RoboDK station: RobotCell.rdk

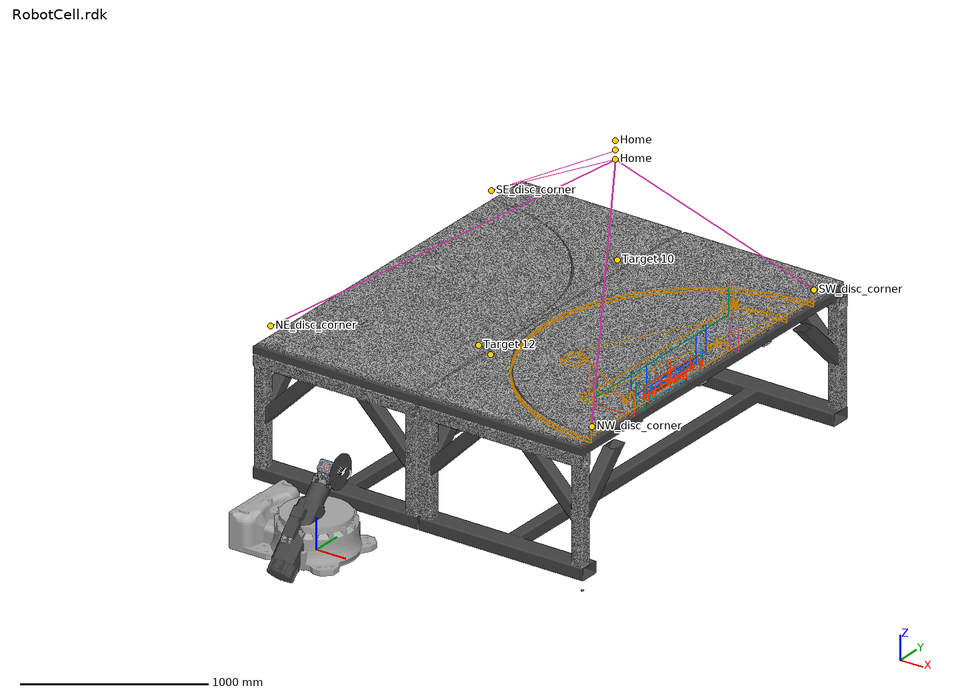
[picture v0: the station drawn from its stored meshes, robots at their saved joint values, targets as dots, program paths as lines]
Station RobotCell (saved by RoboDK 5.6.8). Poses are relative to the parent item; angles as X-Y-Z fixed-axis rotations.
  - frame Kawasaki BX130X Base at (0, 0, 0) mm
    - robot Kawasaki BX130X: 6 axes, payload 130 kg, reach 2991 mm, repeatability 0.06 mm, weight 920 kg
        joint limits [-160, -60, -75, -210, -125, -210] to [160, 76, 90, 210, 125, 210]; home [0, 0, 0, 0, 0, 0]; saved at [15.367, 30.588, 15.611, 20.856, -32.878, -29.669]
      - tool Bare Spindle, TCP at (-2.41, 51.17, 373.7) mm, rotated rx 0.82 ry 46.22 rz 88.69 deg
      - tool Sawblade, TCP at (72.1, 194.8, 514.4) mm, rotated rx 1 ry 44.99 rz 91.98 deg, size 476.9 x 3677.1 x 608 mm, geometry from Sawblade.step
      - tool halfInchUpcut, TCP at (-1.57, 133.94, 455.3) mm, rotated rx 0 ry 45 rz 90 deg, size 451 x 3595 x 525.8 mm, geometry from halfInchUpcut.step
  - frame Work hold down at (0, 0, -2) mm
  - folder FrontWallWest
    - machining project Blade_door_east: C:/Users/kris/AppData/Local/Temp/Front wall cutout v15.apt:2 | rotZ(0) | rotX(0)*rotY(0) | rotz(0) | onStart | onPathStart | onApproach | onPoint | onRetract | onFinish | Extruder(%1) | default | default | OutOnMov(%1) | OutOffMov(%1) | onPathFinish | M_RunCode(%1)
    - machining project Blade_doorframe_east: C:/Users/kris/AppData/Local/Temp/Front wall cutout v15.apt | rotZ(0) | rotX(0)*rotY(0) | rotz(0) | onStart | onPathStart | onApproach | onPoint | onRetract | onFinish | Extruder(%1) | default | default | OutOnMov(%1) | OutOffMov(%1) | onPathFinish | M_RunCode(%1)
    - machining project Blade_doorwindow_east: C:/Users/kris/AppData/Local/Temp/Front wall cutout v11.apt:3 | rotZ(0) | rotX(0)*rotY(0) | rotz(0) | onStart | onPathStart | onApproach | onPoint | onRetract | onFinish | Extruder(%1) | default | default | OutOnMov(%1) | OutOffMov(%1) | onPathFinish | M_RunCode(%1)
    - machining project Blade_door_north: C:/Users/kris/AppData/Local/Temp/Front wall cutout v11.apt:4 | rotZ(0) | rotX(0)*rotY(0) | rotz(0) | onStart | onPathStart | onApproach | onPoint | onRetract | onFinish | Extruder(%1) | default | default | OutOnMov(%1) | OutOffMov(%1) | onPathFinish | M_RunCode(%1)
    - machining project Blade_window_north: C:/Users/kris/AppData/Local/Temp/Front wall cutout v11.apt:5 | rotZ(0) | rotX(0)*rotY(0) | rotz(0) | onStart | onPathStart | onApproach | onPoint | onRetract | onFinish | Extruder(%1) | default | default | OutOnMov(%1) | OutOffMov(%1) | onPathFinish | M_RunCode(%1)
    - machining project Blade_window_south: C:/Users/kris/AppData/Local/Temp/Front wall cutout v11.apt:6 | rotZ(0) | rotX(0)*rotY(0) | rotz(0) | onStart | onPathStart | onApproach | onPoint | onRetract | onFinish | Extruder(%1) | default | default | OutOnMov(%1) | OutOffMov(%1) | onPathFinish | M_RunCode(%1)
    - machining project Roughing: C:/Users/kris/AppData/Local/Temp/Front wall cutout v11.apt:7 | rotZ(0) | rotX(0)*rotY(0) | rotZ(0)
    - machining project Blade_handles_west: C:/Users/kris/AppData/Local/Temp/Front wall cutout v12.apt | rotZ(0) | rotX(0)*rotY(0) | rotz(0) | onStart | onPathStart | onApproach | onPoint | onRetract | onFinish | Extruder(%1) | default | default | OutOnMov(%1) | OutOffMov(%1) | onPathFinish | M_RunCode(%1)
    - machining project Blade_handles_east: C:/Users/kris/AppData/Local/Temp/Front wall cutout v12.apt:2 | rotZ(0) | rotX(0)*rotY(0) | rotz(0) | onStart | onPathStart | onApproach | onPoint | onRetract | onFinish | Extruder(%1) | default | default | OutOnMov(%1) | OutOffMov(%1) | onPathFinish | M_RunCode(%1)
    - machining project Handles_roughing: C:/Users/kris/AppData/Local/Temp/Front wall cutout v12.apt:3 | rotZ(0) | rotX(0)*rotY(0) | rotZ(0) | onStart | onPathStart | onApproach | onPoint | onRetract | onFinish | Extruder(%1) | default | default | OutOnMov(%1) | OutOffMov(%1) | onPathFinish | M_RunCode(%1)
    - program Blade_doorwindow_east (21 instructions, listed below)
    - program Blade_door_north (21 instructions, listed below)
    - program Blade_window_north (21 instructions, listed below)
    - program Blade_window_south (21 instructions, listed below)
    - program Roughing (2440 instructions, listed below)
    - program Blade_handles_west (25 instructions, listed below)
    - program Blade_handles_east (22 instructions, listed below)
    - program Handles_roughing (174 instructions, listed below)
    - program Blade_door_east (20 instructions, listed below)
  - object Front wall cutout v15 at (0, 0, 0) mm, size 2167.6 x 2462.4 x 856 mm, geometry from Front wall cutout v15.step
  - frame CalibrationFrame at (0, 0, 0) mm
    - target Home (Cartesian target) at (0.67, 2769.12, 1198.75) mm, rotated rx -177.74 ry 28.55 rz -88.97 deg; joints [-0.25, 14.674, 2.172, -12.213, -4.012, 10.365] of Kawasaki BX130X
    - target SW_disc_corner (Cartesian target) at (1075.28, 3073.73, 606.29) mm, rotated rx 180 ry 0 rz -88.75 deg; joints [21.99, 63.467, 60.14, 22.667, -46.398, -32.962] of Kawasaki BX130X
    - target Home (Cartesian target) at (0.67, 2769.12, 1198.75) mm, rotated rx -177.74 ry 28.55 rz -88.97 deg; joints [-0.25, 14.674, 2.172, -12.213, -4.012, 10.365] of Kawasaki BX130X
    - target NW_disc_corner (Cartesian target) at (1057.37, 1041.81, 606.29) mm, rotated rx 180 ry 0 rz -88.75 deg; joints [58.442, -29.711, -49.966, 48.514, -54.582, -83.664] of Kawasaki BX130X
    - target Home (Cartesian target) at (0.67, 2769.12, 1198.75) mm, rotated rx -177.74 ry 28.55 rz -88.97 deg; joints [-0.25, 14.674, 2.172, -12.213, -4.012, 10.365] of Kawasaki BX130X
    - target NE_disc_corner (Cartesian target) at (-1038.05, 1060.27, 606.29) mm, rotated rx -180 ry 0 rz -88.75 deg; joints [-56.747, -31.242, -50.944, 132.324, 52.01, -100.14] of Kawasaki BX130X
    - target Home (Cartesian target) at (0.67, 2769.12, 1198.75) mm, rotated rx -177.74 ry 28.55 rz -88.97 deg; joints [-0.25, 14.674, 2.172, -12.213, -4.012, 10.365] of Kawasaki BX130X
    - target SE_disc_corner (Cartesian target) at (-1020.25, 3079.49, 606.29) mm, rotated rx 180 ry 0 rz -88.75 deg; joints [-20.561, 60.823, 55.864, 160.128, 43.451, -151.385] of Kawasaki BX130X
    - target Home (Cartesian target) at (0.67, 2769.12, 1253.75) mm, rotated rx -177.74 ry 28.55 rz -88.97 deg; joints [-0.25, 14.499, 3.862, -8.354, -5.848, 6.491] of Kawasaki BX130X
    - target Target 10 (Cartesian target) at (10.17, 2770.62, 606.29) mm, rotated rx -180 ry 0 rz -90 deg; joints [0.282, 28.794, 8.219, 0.482, -24.427, -0.639] of Kawasaki BX130X
    - target Home (Cartesian target) at (0.67, 2769.12, 1253.75) mm, rotated rx -177.74 ry 28.55 rz -88.97 deg; joints [-0.25, 14.499, 3.862, -8.354, -5.848, 6.491] of Kawasaki BX130X
    - target Target 12 (Cartesian target) at (-1.2, 1504.96, 606.29) mm, rotated rx 180 ry 0 rz -88.97 deg; joints [0.375, -38.885, -55.483, 2.09, -28.427, -2.833] of Kawasaki BX130X
    - target Home (Cartesian target) at (0.67, 2769.12, 1308.75) mm, rotated rx -177.74 ry 28.55 rz -88.97 deg; joints [-0.25, 14.413, 5.654, -6.334, -7.711, 4.458] of Kawasaki BX130X
    - target Target 14 (Cartesian target) at (114.89, 1450.3, 606.29) mm, rotated rx 180 ry 0 rz -88.97 deg; joints [6.616, -42.397, -57.387, 10.621, -30.699, -14.583] of Kawasaki BX130X
  - program checkTableCalibration (11 instructions, listed below)
  - program Blade_doorframe_east (24 instructions, listed below)
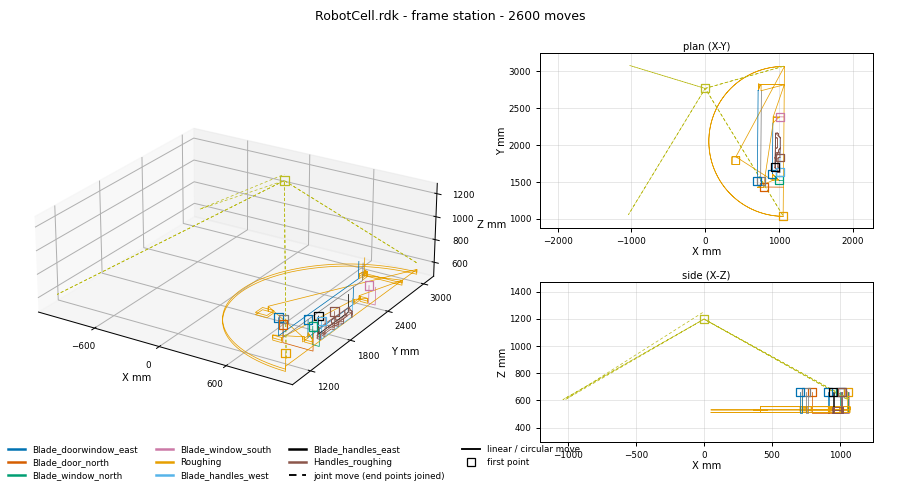
[picture p0: tool path of RobotCell.rdk in frame station, 2600 of 2600 moves have a stored position in this frame; points joined in program order, loops and branches not executed]

--- program Blade_doorwindow_east (robot Kawasaki BX130X) ---
  Smooth(1)
  Set speed (100.0 mm/s)
  Set Ref.: Work hold down
  Set Tool: Sawblade
  Show Sawblade
  MoveJ 1 to (911.47, 1609.21, 666.29) mm, rotated rx 180 ry 0 rz -90.5 deg; joints [34.508, -17.696, -36.382, 39.95, -39.175, -59.907]
  MoveL 2 to (911.47, 1609.21, 666.29) mm, rotated rx 180 ry 0 rz -90.5 deg; joints [34.508, -17.696, -36.382, 39.95, -39.175, -59.907]
  MoveL 3 to (911.47, 1609.21, 566.29) mm, rotated rx 180 ry 0 rz -90.5 deg; joints [34.508, -16.451, -38.924, 43.196, -36.34, -64.01]
  MoveL 4 to (911.47, 1609.21, 566.29) mm, rotated rx 180 ry 0 rz -90.5 deg; joints [34.508, -16.451, -38.924, 43.196, -36.34, -64.01]
  Set speed (100.0 mm/s)
  MoveL 5 to (911.47, 1609.21, 556.29) mm, rotated rx -180 ry 0 rz -90.5 deg; joints [34.508, -16.304, -39.162, 43.558, -36.06, -64.458]
  Set speed (5.6 mm/s)
  MoveL 6 to (911.47, 1609.21, 551.89) mm, rotated rx -180 ry 0 rz -90.5 deg; joints [34.508, -16.239, -39.266, 43.719, -35.937, -64.658]
  MoveL 7 to (911.47, 1609.21, 513.19) mm, rotated rx 180 ry 0 rz -90.5 deg; joints [34.508, -15.625, -40.158, 45.203, -34.863, -66.478]
  Set speed (133.3 mm/s)
  MoveL 8 to (917.55, 2299.44, 513.19) mm, rotated rx -180 ry 0 rz -90.5 deg; joints [23.876, 14.834, -9.851, 37.999, -28.292, -52.853]
  Set speed (100.0 mm/s)
  MoveL 9 to (917.55, 2299.44, 566.29) mm, rotated rx -180 ry 0 rz -90.5 deg; joints [23.876, 14.117, -8.799, 36.076, -29.704, -50.655]
  MoveL 10 to (917.55, 2299.44, 566.29) mm, rotated rx -180 ry 0 rz -90.5 deg; joints [23.876, 14.117, -8.799, 36.076, -29.704, -50.655]
  MoveL 11 to (917.55, 2299.44, 666.29) mm, rotated rx 180 ry 0 rz -90.5 deg; joints [23.876, 12.98, -6.592, 32.933, -32.461, -46.986]
  Print: /'Blade door top'

--- program Blade_door_north (robot Kawasaki BX130X) ---
  Smooth(1)
  Set speed (100.0 mm/s)
  Set Ref.: Work hold down
  Set Tool: Sawblade
  Show Sawblade
  MoveJ 1 to (794.89, 1433.16, 666.29) mm, rotated rx -180 ry 0 rz 179.5 deg; joints [15.202, -13.662, -33.122, -48.467, -65.42, 92.913]
  MoveL 2 to (794.89, 1433.16, 666.29) mm, rotated rx -180 ry 0 rz 179.5 deg; joints [15.202, -13.662, -33.122, -48.467, -65.42, 92.913]
  MoveL 3 to (794.89, 1433.16, 566.29) mm, rotated rx 180 ry 0 rz 179.5 deg; joints [15.202, -12.385, -35.587, -49.836, -62.972, 96.057]
  MoveL 4 to (794.89, 1433.16, 566.29) mm, rotated rx 180 ry 0 rz 179.5 deg; joints [15.202, -12.385, -35.587, -49.836, -62.972, 96.057]
  Set speed (100.0 mm/s)
  MoveL 5 to (794.89, 1433.16, 556.29) mm, rotated rx -180 ry 0 rz 179.5 deg; joints [15.202, -12.236, -35.818, -49.985, -62.728, 96.384]
  Set speed (5.6 mm/s)
  MoveL 6 to (794.89, 1433.16, 551.89) mm, rotated rx -180 ry 0 rz 179.5 deg; joints [15.202, -12.169, -35.918, -50.052, -62.62, 96.528]
  MoveL 7 to (794.89, 1433.16, 513.19) mm, rotated rx -180 ry 0 rz 179.5 deg; joints [15.202, -11.55, -36.78, -50.654, -61.675, 97.818]
  Set speed (133.3 mm/s)
  MoveL 8 to (1060.8, 1430.82, 513.19) mm, rotated rx -180 ry 0 rz 179.5 deg; joints [24.193, -6.922, -32.695, -51.648, -55.011, 92.337]
  Set speed (100.0 mm/s)
  MoveL 9 to (1060.8, 1430.82, 566.29) mm, rotated rx -180 ry 0 rz 179.5 deg; joints [24.193, -7.755, -31.542, -50.591, -56.258, 90.464]
  MoveL 10 to (1060.8, 1430.82, 566.29) mm, rotated rx -180 ry 0 rz 179.5 deg; joints [24.193, -7.755, -31.542, -50.591, -56.258, 90.464]
  MoveL 11 to (1060.8, 1430.82, 666.29) mm, rotated rx -180 ry 0 rz 179.5 deg; joints [24.193, -9.049, -29.155, -48.799, -58.64, 87.134]
  Print: /'Blade door window top'

--- program Blade_window_north (robot Kawasaki BX130X) ---
  Smooth(1)
  Set speed (100.0 mm/s)
  Set Ref.: Work hold down
  Set Tool: Sawblade
  Show Sawblade
  MoveJ 1 to (1002.24, 1523.24, 666.29) mm, rotated rx -180 ry 0 rz 179.5 deg; joints [21.13, -5.832, -26.235, -48.977, -60.608, 89.581]
  MoveL 2 to (1002.24, 1523.24, 666.29) mm, rotated rx -180 ry 0 rz 179.5 deg; joints [21.13, -5.832, -26.235, -48.977, -60.608, 89.581]
  MoveL 3 to (1002.24, 1523.24, 566.29) mm, rotated rx -180 ry 0 rz 179.5 deg; joints [21.13, -4.54, -28.576, -50.616, -58.262, 92.804]
  MoveL 4 to (1002.24, 1523.24, 566.29) mm, rotated rx -180 ry 0 rz 179.5 deg; joints [21.13, -4.54, -28.576, -50.616, -58.262, 92.804]
  Set speed (100.0 mm/s)
  MoveL 5 to (1002.24, 1523.24, 556.29) mm, rotated rx -180 ry 0 rz 179.5 deg; joints [21.13, -4.392, -28.794, -50.793, -58.03, 93.138]
  Set speed (5.6 mm/s)
  MoveL 6 to (1002.24, 1523.24, 551.89) mm, rotated rx 180 ry 0 rz 179.5 deg; joints [21.13, -4.325, -28.89, -50.871, -57.928, 93.286]
  MoveL 7 to (1002.24, 1523.24, 513.19) mm, rotated rx -180 ry 0 rz 179.5 deg; joints [21.13, -3.713, -29.703, -51.58, -57.035, 94.604]
  Set speed (133.3 mm/s)
  MoveL 8 to (1061.61, 1522.72, 513.19) mm, rotated rx 180 ry 0 rz 179.5 deg; joints [22.97, -2.615, -28.649, -51.728, -55.71, 93.414]
  Set speed (100.0 mm/s)
  MoveL 9 to (1061.61, 1522.72, 566.29) mm, rotated rx 180 ry 0 rz 179.5 deg; joints [22.97, -3.438, -27.529, -50.718, -56.927, 91.594]
  MoveL 10 to (1061.61, 1522.72, 566.29) mm, rotated rx 180 ry 0 rz 179.5 deg; joints [22.97, -3.438, -27.529, -50.718, -56.927, 91.594]
  MoveL 11 to (1061.61, 1522.72, 666.29) mm, rotated rx 180 ry 0 rz 179.5 deg; joints [22.97, -4.728, -25.203, -48.996, -59.259, 88.337]
  Print: /'Blade door window south'

--- program Blade_window_south (robot Kawasaki BX130X) ---
  Smooth(1)
  Set speed (100.0 mm/s)
  Set Ref.: Work hold down
  Set Tool: Sawblade
  Show Sawblade
  MoveJ 1 to (1009.82, 2383.81, 666.29) mm, rotated rx -180 ry 0 rz 179.49 deg; joints [14.255, 35.484, 22.375, -46.548, -70.389, 88.528]
  MoveL 2 to (1009.82, 2383.81, 666.29) mm, rotated rx -180 ry 0 rz 179.49 deg; joints [14.255, 35.484, 22.375, -46.548, -70.389, 88.528]
  MoveL 3 to (1009.82, 2383.81, 566.29) mm, rotated rx -180 ry 0 rz 179.49 deg; joints [14.255, 36.15, 19.85, -47.43, -68.212, 91.022]
  MoveL 4 to (1009.82, 2383.81, 566.29) mm, rotated rx -180 ry 0 rz 179.49 deg; joints [14.255, 36.15, 19.85, -47.43, -68.212, 91.022]
  Set speed (100.0 mm/s)
  MoveL 5 to (1009.82, 2383.81, 556.29) mm, rotated rx -180 ry 0 rz 179.49 deg; joints [14.255, 36.232, 19.62, -47.522, -68, 91.271]
  Set speed (5.6 mm/s)
  MoveL 6 to (1009.82, 2383.81, 551.89) mm, rotated rx -180 ry 0 rz 179.49 deg; joints [14.255, 36.27, 19.519, -47.563, -67.907, 91.381]
  MoveL 7 to (1009.82, 2383.81, 513.19) mm, rotated rx -180 ry 0 rz 179.49 deg; joints [14.255, 36.621, 18.668, -47.932, -67.099, 92.344]
  Set speed (133.3 mm/s)
  MoveL 8 to (1069.19, 2383.28, 513.19) mm, rotated rx -180 ry 0 rz 179.49 deg; joints [15.552, 37.428, 19.819, -47.863, -66.413, 91.165]
  Set speed (100.0 mm/s)
  MoveL 9 to (1069.19, 2383.28, 566.29) mm, rotated rx 180 ry 0 rz 179.49 deg; joints [15.552, 36.97, 21.014, -47.344, -67.527, 89.838]
  MoveL 10 to (1069.19, 2383.28, 566.29) mm, rotated rx 180 ry 0 rz 179.49 deg; joints [15.552, 36.97, 21.014, -47.344, -67.527, 89.838]
  MoveL 11 to (1069.19, 2383.28, 666.29) mm, rotated rx -180 ry 0 rz 179.49 deg; joints [15.552, 36.33, 23.568, -46.431, -69.711, 87.335]
  Print: /'Roughing'

--- program Roughing (robot Kawasaki BX130X) ---
  Smooth(1)
  Set speed (100.0 mm/s)
  Set Ref.: Work hold down
  Set Tool: halfInchUpcut
  Show halfInchUpcut
  MoveJ 1 to (1057.31, 1035.46, 666.29) mm, rotated rx -180 ry 0 rz -88.32 deg; joints [58.753, -30.506, -48.445, 47.413, -56.648, -82.141]
  MoveL 2 to (1057.31, 1035.46, 666.29) mm, rotated rx -180 ry 0 rz -88.32 deg; joints [58.753, -30.506, -48.445, 47.413, -56.648, -82.141]
  MoveL 3 to (1057.31, 1035.46, 566.29) mm, rotated rx 180 ry 0 rz -88.32 deg; joints [58.753, -29.128, -51.071, 49.488, -53.99, -85.786]
  MoveL 4 to (1057.31, 1035.46, 566.29) mm, rotated rx 180 ry 0 rz -88.32 deg; joints [58.753, -29.128, -51.071, 49.488, -53.99, -85.786]
  Set speed (100.0 mm/s)
  MoveL 5 to (1057.31, 1035.46, 556.29) mm, rotated rx -180 ry 0 rz -88.32 deg; joints [58.753, -28.961, -51.317, 49.718, -53.723, -86.175]
  Set speed (5.6 mm/s)
  MoveL 6 to (1057.31, 1035.46, 552.29) mm, rotated rx -180 ry 0 rz -88.32 deg; joints [58.753, -28.893, -51.415, 49.811, -53.616, -86.332]
  MoveL 7 to (1057.31, 1035.46, 532.29) mm, rotated rx 180 ry 0 rz -88.32 deg; joints [58.753, -28.539, -51.896, 50.287, -53.08, -87.13]
  Set speed (91.9 mm/s)
  MoveL 8 to (1054.46, 1035.49, 532.29) mm, rotated rx 180 ry 0 rz -88.32 deg; joints [58.684, -28.699, -52.001, 50.252, -53.066, -87.026]
  MoveL 9 to (1051.61, 1035.53, 532.29) mm, rotated rx -180 ry 0 rz -88.32 deg; joints [58.614, -28.86, -52.105, 50.217, -53.053, -86.921]
  MoveL 10 to (1048.77, 1035.57, 532.29) mm, rotated rx 180 ry 0 rz -88.32 deg; joints [58.544, -29.02, -52.209, 50.181, -53.039, -86.816]
  MoveL 11 to (1045.92, 1035.62, 532.29) mm, rotated rx -180 ry 0 rz -88.32 deg; joints [58.473, -29.18, -52.313, 50.145, -53.025, -86.71]
  MoveL 12 to (1043.07, 1035.69, 532.29) mm, rotated rx -180 ry 0 rz -88.32 deg; joints [58.402, -29.34, -52.417, 50.109, -53.011, -86.603]
  MoveL 13 to (1040.22, 1035.75, 532.29) mm, rotated rx -180 ry 0 rz -88.32 deg; joints [58.33, -29.5, -52.52, 50.072, -52.997, -86.495]
  MoveL 14 to (1037.37, 1035.83, 532.29) mm, rotated rx -180 ry 0 rz -88.32 deg; joints [58.258, -29.659, -52.623, 50.035, -52.982, -86.387]
  MoveL 15 to (1034.52, 1035.92, 532.29) mm, rotated rx -180 ry 0 rz -88.32 deg; joints [58.185, -29.819, -52.726, 49.998, -52.967, -86.278]
  MoveL 16 to (1031.67, 1036.01, 532.29) mm, rotated rx 180 ry 0 rz -88.32 deg; joints [58.111, -29.978, -52.828, 49.961, -52.952, -86.169]
  MoveL 17 to (1028.82, 1036.11, 532.29) mm, rotated rx 180 ry 0 rz -88.32 deg; joints [58.037, -30.138, -52.93, 49.923, -52.937, -86.058]
  MoveL 18 to (1025.98, 1036.22, 532.29) mm, rotated rx 180 ry 0 rz -88.32 deg; joints [57.962, -30.297, -53.031, 49.885, -52.921, -85.947]
  MoveL 19 to (1023.13, 1036.34, 532.29) mm, rotated rx 180 ry 0 rz -88.32 deg; joints [57.887, -30.456, -53.132, 49.847, -52.906, -85.836]
  MoveL 20 to (1020.28, 1036.46, 532.29) mm, rotated rx -180 ry 0 rz -88.32 deg; joints [57.811, -30.615, -53.233, 49.808, -52.889, -85.723]
  MoveL 21 to (1017.43, 1036.6, 532.29) mm, rotated rx 180 ry 0 rz -88.32 deg; joints [57.734, -30.774, -53.334, 49.769, -52.873, -85.61]
  MoveL 22 to (1014.59, 1036.74, 532.29) mm, rotated rx -180 ry 0 rz -88.32 deg; joints [57.657, -30.933, -53.434, 49.73, -52.857, -85.496]
  MoveL 23 to (1011.74, 1036.89, 532.29) mm, rotated rx -180 ry 0 rz -88.32 deg; joints [57.579, -31.092, -53.534, 49.691, -52.84, -85.381]
  MoveL 24 to (1008.9, 1037.04, 532.29) mm, rotated rx -180 ry 0 rz -88.32 deg; joints [57.501, -31.25, -53.633, 49.651, -52.823, -85.266]
  MoveL 25 to (1006.05, 1037.21, 532.29) mm, rotated rx -180 ry 0 rz -88.32 deg; joints [57.422, -31.409, -53.733, 49.611, -52.805, -85.15]
  MoveL 26 to (1003.21, 1037.38, 532.29) mm, rotated rx 180 ry 0 rz -88.32 deg; joints [57.342, -31.567, -53.831, 49.57, -52.788, -85.033]
  MoveL 27 to (1000.36, 1037.56, 532.29) mm, rotated rx -180 ry 0 rz -88.32 deg; joints [57.262, -31.725, -53.93, 49.53, -52.77, -84.916]
  MoveL 28 to (997.52, 1037.75, 532.29) mm, rotated rx -180 ry 0 rz -88.32 deg; joints [57.181, -31.883, -54.028, 49.489, -52.752, -84.798]
  MoveL 29 to (994.68, 1037.95, 532.29) mm, rotated rx -180 ry 0 rz -88.32 deg; joints [57.099, -32.04, -54.126, 49.447, -52.733, -84.679]
  MoveL 30 to (991.83, 1038.15, 532.29) mm, rotated rx -180 ry 0 rz -88.32 deg; joints [57.017, -32.198, -54.223, 49.406, -52.715, -84.559]
  MoveL 31 to (988.99, 1038.36, 532.29) mm, rotated rx 180 ry 0 rz -88.32 deg; joints [56.935, -32.355, -54.32, 49.364, -52.696, -84.439]
  MoveL 32 to (986.15, 1038.58, 532.29) mm, rotated rx 180 ry 0 rz -88.32 deg; joints [56.851, -32.512, -54.417, 49.322, -52.676, -84.318]
  MoveL 33 to (983.31, 1038.81, 532.29) mm, rotated rx 180 ry 0 rz -88.32 deg; joints [56.767, -32.669, -54.513, 49.279, -52.657, -84.196]
  MoveL 34 to (980.47, 1039.05, 532.29) mm, rotated rx -180 ry 0 rz -88.32 deg; joints [56.683, -32.826, -54.609, 49.236, -52.637, -84.074]
  MoveL 35 to (977.63, 1039.29, 532.29) mm, rotated rx 180 ry 0 rz -88.32 deg; joints [56.598, -32.982, -54.704, 49.193, -52.617, -83.951]
  MoveL 36 to (974.79, 1039.55, 532.29) mm, rotated rx 180 ry 0 rz -88.32 deg; joints [56.512, -33.139, -54.8, 49.15, -52.597, -83.827]
  MoveL 37 to (971.95, 1039.81, 532.29) mm, rotated rx 180 ry 0 rz -88.32 deg; joints [56.425, -33.295, -54.894, 49.106, -52.576, -83.702]
  MoveL 38 to (969.12, 1040.08, 532.29) mm, rotated rx -180 ry 0 rz -88.32 deg; joints [56.338, -33.451, -54.989, 49.062, -52.555, -83.577]
  MoveL 39 to (966.28, 1040.35, 532.29) mm, rotated rx -180 ry 0 rz -88.32 deg; joints [56.251, -33.606, -55.083, 49.017, -52.534, -83.451]
  MoveL 40 to (963.44, 1040.64, 532.29) mm, rotated rx 180 ry 0 rz -88.32 deg; joints [56.162, -33.762, -55.176, 48.973, -52.512, -83.325]
  MoveL 41 to (960.61, 1040.93, 532.29) mm, rotated rx -180 ry 0 rz -88.32 deg; joints [56.073, -33.917, -55.27, 48.928, -52.49, -83.197]
  MoveL 42 to (957.78, 1041.23, 532.29) mm, rotated rx -180 ry 0 rz -88.32 deg; joints [55.984, -34.072, -55.363, 48.882, -52.468, -83.069]
  MoveL 43 to (954.94, 1041.54, 532.29) mm, rotated rx 180 ry 0 rz -88.32 deg; joints [55.894, -34.226, -55.455, 48.836, -52.446, -82.94]
  MoveL 44 to (952.11, 1041.85, 532.29) mm, rotated rx 180 ry 0 rz -88.32 deg; joints [55.803, -34.381, -55.547, 48.79, -52.423, -82.811]
  MoveL 45 to (949.28, 1042.18, 532.29) mm, rotated rx 180 ry 0 rz -88.32 deg; joints [55.711, -34.535, -55.639, 48.744, -52.4, -82.681]
  MoveL 46 to (946.45, 1042.51, 532.29) mm, rotated rx 180 ry 0 rz -88.32 deg; joints [55.619, -34.688, -55.73, 48.697, -52.376, -82.55]
  MoveL 47 to (943.62, 1042.85, 532.29) mm, rotated rx -180 ry 0 rz -88.32 deg; joints [55.526, -34.842, -55.821, 48.65, -52.353, -82.418]
  MoveL 48 to (940.79, 1043.2, 532.29) mm, rotated rx -180 ry 0 rz -88.32 deg; joints [55.433, -34.995, -55.912, 48.603, -52.329, -82.286]
  MoveL 49 to (937.96, 1043.56, 532.29) mm, rotated rx -180 ry 0 rz -88.32 deg; joints [55.339, -35.148, -56.002, 48.555, -52.304, -82.153]
  MoveL 50 to (935.14, 1043.92, 532.29) mm, rotated rx 180 ry 0 rz -88.32 deg; joints [55.244, -35.301, -56.092, 48.507, -52.28, -82.02]
  MoveL 51 to (932.31, 1044.29, 532.29) mm, rotated rx -180 ry 0 rz -88.32 deg; joints [55.149, -35.453, -56.181, 48.458, -52.255, -81.885]
  MoveL 52 to (929.49, 1044.67, 532.29) mm, rotated rx -180 ry 0 rz -88.32 deg; joints [55.053, -35.605, -56.27, 48.41, -52.229, -81.75]
  MoveL 53 to (926.66, 1045.06, 532.29) mm, rotated rx -180 ry 0 rz -88.32 deg; joints [54.956, -35.757, -56.358, 48.361, -52.204, -81.615]
  MoveL 54 to (923.84, 1045.45, 532.29) mm, rotated rx -180 ry 0 rz -88.32 deg; joints [54.859, -35.908, -56.447, 48.311, -52.178, -81.478]
  MoveL 55 to (921.02, 1045.86, 532.29) mm, rotated rx 180 ry 0 rz -88.32 deg; joints [54.761, -36.059, -56.534, 48.261, -52.151, -81.341]
  MoveL 56 to (918.2, 1046.27, 532.29) mm, rotated rx 180 ry 0 rz -88.32 deg; joints [54.663, -36.21, -56.622, 48.211, -52.125, -81.203]
  MoveL 57 to (915.38, 1046.69, 532.29) mm, rotated rx 180 ry 0 rz -88.32 deg; joints [54.563, -36.36, -56.708, 48.161, -52.098, -81.065]
  MoveL 58 to (912.56, 1047.11, 532.29) mm, rotated rx 180 ry 0 rz -88.32 deg; joints [54.464, -36.51, -56.795, 48.11, -52.07, -80.926]
  MoveL 59 to (909.75, 1047.55, 532.29) mm, rotated rx 180 ry 0 rz -88.32 deg; joints [54.363, -36.659, -56.881, 48.059, -52.043, -80.786]
  MoveL 60 to (906.93, 1047.99, 532.29) mm, rotated rx 180 ry 0 rz -88.32 deg; joints [54.262, -36.809, -56.967, 48.007, -52.015, -80.646]
  MoveL 61 to (904.12, 1048.44, 532.29) mm, rotated rx -180 ry 0 rz -88.32 deg; joints [54.16, -36.957, -57.052, 47.955, -51.986, -80.504]
  MoveL 62 to (901.31, 1048.9, 532.29) mm, rotated rx 180 ry 0 rz -88.32 deg; joints [54.058, -37.106, -57.136, 47.903, -51.957, -80.363]
  MoveL 63 to (898.49, 1049.37, 532.29) mm, rotated rx -180 ry 0 rz -88.32 deg; joints [53.955, -37.254, -57.221, 47.851, -51.928, -80.22]
  MoveL 64 to (895.68, 1049.84, 532.29) mm, rotated rx -180 ry 0 rz -88.32 deg; joints [53.851, -37.401, -57.305, 47.798, -51.899, -80.077]
  MoveL 65 to (892.87, 1050.33, 532.29) mm, rotated rx 180 ry 0 rz -88.32 deg; joints [53.747, -37.549, -57.388, 47.744, -51.869, -79.933]
  MoveL 66 to (890.07, 1050.82, 532.29) mm, rotated rx -180 ry 0 rz -88.32 deg; joints [53.641, -37.695, -57.471, 47.691, -51.839, -79.789]
  MoveL 67 to (887.26, 1051.31, 532.29) mm, rotated rx 180 ry 0 rz -88.32 deg; joints [53.536, -37.842, -57.554, 47.637, -51.808, -79.643]
  MoveL 68 to (884.46, 1051.82, 532.29) mm, rotated rx 180 ry 0 rz -88.32 deg; joints [53.429, -37.988, -57.636, 47.582, -51.777, -79.497]
  MoveL 69 to (881.65, 1052.33, 532.29) mm, rotated rx 180 ry 0 rz -88.32 deg; joints [53.322, -38.133, -57.718, 47.527, -51.746, -79.351]
  MoveL 70 to (878.85, 1052.86, 532.29) mm, rotated rx -180 ry 0 rz -88.32 deg; joints [53.215, -38.278, -57.799, 47.472, -51.714, -79.204]
  MoveL 71 to (876.05, 1053.39, 532.29) mm, rotated rx 180 ry 0 rz -88.32 deg; joints [53.106, -38.422, -57.88, 47.417, -51.682, -79.056]
  MoveL 72 to (873.25, 1053.92, 532.29) mm, rotated rx 180 ry 0 rz -88.32 deg; joints [52.998, -38.567, -57.96, 47.361, -51.649, -78.908]
  MoveL 73 to (870.46, 1054.47, 532.29) mm, rotated rx -180 ry 0 rz -88.32 deg; joints [52.888, -38.71, -58.04, 47.305, -51.617, -78.758]
  MoveL 74 to (867.66, 1055.02, 532.29) mm, rotated rx -180 ry 0 rz -88.32 deg; joints [52.778, -38.853, -58.119, 47.248, -51.583, -78.609]
  MoveL 75 to (864.87, 1055.58, 532.29) mm, rotated rx -180 ry 0 rz -88.32 deg; joints [52.667, -38.996, -58.198, 47.191, -51.55, -78.458]
  MoveL 76 to (862.07, 1056.15, 532.29) mm, rotated rx 180 ry 0 rz -88.32 deg; joints [52.555, -39.138, -58.277, 47.134, -51.516, -78.307]
  MoveL 77 to (859.28, 1056.73, 532.29) mm, rotated rx -180 ry 0 rz -88.32 deg; joints [52.443, -39.279, -58.355, 47.076, -51.481, -78.156]
  MoveL 78 to (856.49, 1057.31, 532.29) mm, rotated rx 180 ry 0 rz -88.32 deg; joints [52.33, -39.42, -58.432, 47.018, -51.446, -78.003]
  MoveL 79 to (853.71, 1057.91, 532.29) mm, rotated rx 180 ry 0 rz -88.32 deg; joints [52.217, -39.561, -58.509, 46.96, -51.411, -77.85]
  MoveL 80 to (850.92, 1058.51, 532.29) mm, rotated rx 180 ry 0 rz -88.32 deg; joints [52.102, -39.701, -58.586, 46.901, -51.375, -77.697]
  MoveL 81 to (848.14, 1059.11, 532.29) mm, rotated rx -180 ry 0 rz -88.32 deg; joints [51.988, -39.84, -58.662, 46.842, -51.339, -77.543]
  MoveL 82 to (845.35, 1059.73, 532.29) mm, rotated rx -180 ry 0 rz -88.32 deg; joints [51.872, -39.979, -58.738, 46.782, -51.303, -77.388]
  MoveL 83 to (842.57, 1060.35, 532.29) mm, rotated rx -180 ry 0 rz -88.32 deg; joints [51.756, -40.118, -58.813, 46.722, -51.266, -77.232]
  MoveL 84 to (839.79, 1060.98, 532.29) mm, rotated rx -180 ry 0 rz -88.32 deg; joints [51.639, -40.255, -58.888, 46.662, -51.229, -77.076]
  MoveL 85 to (837.02, 1061.62, 532.29) mm, rotated rx 180 ry 0 rz -88.32 deg; joints [51.522, -40.393, -58.962, 46.601, -51.191, -76.919]
  MoveL 86 to (834.24, 1062.27, 532.29) mm, rotated rx -180 ry 0 rz -88.32 deg; joints [51.404, -40.529, -59.036, 46.54, -51.153, -76.762]
  MoveL 87 to (831.47, 1062.93, 532.29) mm, rotated rx 180 ry 0 rz -88.32 deg; joints [51.285, -40.665, -59.109, 46.479, -51.114, -76.604]
  MoveL 88 to (828.7, 1063.59, 532.29) mm, rotated rx 180 ry 0 rz -88.32 deg; joints [51.166, -40.8, -59.182, 46.417, -51.075, -76.446]
  MoveL 89 to (825.93, 1064.26, 532.29) mm, rotated rx -180 ry 0 rz -88.32 deg; joints [51.046, -40.935, -59.255, 46.354, -51.036, -76.287]
  MoveL 90 to (823.16, 1064.94, 532.29) mm, rotated rx -180 ry 0 rz -88.32 deg; joints [50.925, -41.069, -59.326, 46.292, -50.996, -76.127]
  MoveL 91 to (820.39, 1065.62, 532.29) mm, rotated rx 180 ry 0 rz -88.32 deg; joints [50.804, -41.203, -59.398, 46.229, -50.956, -75.967]
  MoveL 92 to (817.63, 1066.32, 532.29) mm, rotated rx 180 ry 0 rz -88.32 deg; joints [50.682, -41.336, -59.469, 46.165, -50.915, -75.806]
  MoveL 93 to (814.86, 1067.02, 532.29) mm, rotated rx 180 ry 0 rz -88.32 deg; joints [50.559, -41.468, -59.539, 46.102, -50.874, -75.644]
  MoveL 94 to (812.1, 1067.73, 532.29) mm, rotated rx -180 ry 0 rz -88.32 deg; joints [50.436, -41.599, -59.609, 46.037, -50.832, -75.482]
  MoveL 95 to (809.35, 1068.44, 532.29) mm, rotated rx -180 ry 0 rz -88.32 deg; joints [50.312, -41.73, -59.678, 45.973, -50.79, -75.319]
  MoveL 96 to (806.59, 1069.17, 532.29) mm, rotated rx 180 ry 0 rz -88.32 deg; joints [50.188, -41.86, -59.747, 45.908, -50.748, -75.156]
  MoveL 97 to (803.84, 1069.9, 532.29) mm, rotated rx 180 ry 0 rz -88.32 deg; joints [50.063, -41.99, -59.815, 45.843, -50.705, -74.992]
  MoveL 98 to (801.08, 1070.64, 532.29) mm, rotated rx -180 ry 0 rz -88.32 deg; joints [49.937, -42.119, -59.883, 45.777, -50.662, -74.828]
  MoveL 99 to (798.33, 1071.39, 532.29) mm, rotated rx 180 ry 0 rz -88.32 deg; joints [49.811, -42.247, -59.95, 45.711, -50.618, -74.663]
  MoveL 100 to (795.59, 1072.14, 532.29) mm, rotated rx 180 ry 0 rz -88.32 deg; joints [49.684, -42.374, -60.017, 45.644, -50.574, -74.497]
  MoveL 101 to (792.84, 1072.91, 532.29) mm, rotated rx 180 ry 0 rz -88.32 deg; joints [49.556, -42.501, -60.084, 45.577, -50.529, -74.331]
  MoveL 102 to (790.1, 1073.68, 532.29) mm, rotated rx 180 ry 0 rz -88.32 deg; joints [49.428, -42.627, -60.149, 45.51, -50.484, -74.165]
  MoveL 103 to (787.35, 1074.45, 532.29) mm, rotated rx -180 ry 0 rz -88.32 deg; joints [49.299, -42.752, -60.215, 45.442, -50.438, -73.998]
  MoveL 104 to (784.62, 1075.24, 532.29) mm, rotated rx -180 ry 0 rz -88.32 deg; joints [49.169, -42.876, -60.279, 45.374, -50.392, -73.83]
  MoveL 105 to (781.88, 1076.03, 532.29) mm, rotated rx 180 ry 0 rz -88.32 deg; joints [49.039, -43, -60.343, 45.306, -50.345, -73.662]
  MoveL 106 to (779.14, 1076.84, 532.29) mm, rotated rx 180 ry 0 rz -88.32 deg; joints [48.908, -43.123, -60.407, 45.237, -50.298, -73.493]
  MoveL 107 to (776.41, 1077.65, 532.29) mm, rotated rx 180 ry 0 rz -88.32 deg; joints [48.777, -43.245, -60.47, 45.168, -50.251, -73.324]
  MoveL 108 to (773.68, 1078.46, 532.29) mm, rotated rx 180 ry 0 rz -88.32 deg; joints [48.645, -43.366, -60.533, 45.098, -50.203, -73.154]
  MoveL 109 to (770.95, 1079.29, 532.29) mm, rotated rx -180 ry 0 rz -88.32 deg; joints [48.512, -43.487, -60.595, 45.028, -50.155, -72.983]
  MoveL 110 to (768.23, 1080.12, 532.29) mm, rotated rx 180 ry 0 rz -88.32 deg; joints [48.379, -43.606, -60.656, 44.958, -50.106, -72.812]
  MoveL 111 to (765.5, 1080.96, 532.29) mm, rotated rx -180 ry 0 rz -88.32 deg; joints [48.245, -43.725, -60.717, 44.887, -50.056, -72.641]
  MoveL 112 to (762.78, 1081.81, 532.29) mm, rotated rx 180 ry 0 rz -88.32 deg; joints [48.111, -43.843, -60.778, 44.816, -50.007, -72.469]
  MoveL 113 to (760.06, 1082.66, 532.29) mm, rotated rx -180 ry 0 rz -88.32 deg; joints [47.976, -43.961, -60.838, 44.744, -49.956, -72.297]
  MoveL 114 to (757.35, 1083.52, 532.29) mm, rotated rx 180 ry 0 rz -88.32 deg; joints [47.84, -44.077, -60.897, 44.672, -49.905, -72.124]
  MoveL 115 to (754.63, 1084.39, 532.29) mm, rotated rx -180 ry 0 rz -88.32 deg; joints [47.704, -44.192, -60.956, 44.6, -49.854, -71.95]
  MoveL 116 to (751.92, 1085.27, 532.29) mm, rotated rx 180 ry 0 rz -88.32 deg; joints [47.567, -44.307, -61.014, 44.527, -49.802, -71.776]
  MoveL 117 to (749.21, 1086.16, 532.29) mm, rotated rx 180 ry 0 rz -88.32 deg; joints [47.43, -44.421, -61.072, 44.454, -49.75, -71.602]
  MoveL 118 to (746.51, 1087.05, 532.29) mm, rotated rx -180 ry 0 rz -88.32 deg; joints [47.292, -44.534, -61.129, 44.38, -49.697, -71.427]
  MoveL 119 to (743.8, 1087.95, 532.29) mm, rotated rx 180 ry 0 rz -88.32 deg; joints [47.153, -44.646, -61.186, 44.306, -49.644, -71.252]
  MoveL 120 to (741.1, 1088.86, 532.29) mm, rotated rx 180 ry 0 rz -88.32 deg; joints [47.014, -44.757, -61.242, 44.232, -49.59, -71.076]
  MoveL 121 to (738.4, 1089.78, 532.29) mm, rotated rx -180 ry 0 rz -88.32 deg; joints [46.875, -44.867, -61.297, 44.157, -49.536, -70.9]
  MoveL 122 to (735.71, 1090.7, 532.29) mm, rotated rx -180 ry 0 rz -88.32 deg; joints [46.734, -44.976, -61.352, 44.082, -49.481, -70.723]
  MoveL 123 to (733.01, 1091.63, 532.29) mm, rotated rx 180 ry 0 rz -88.32 deg; joints [46.593, -45.084, -61.407, 44.006, -49.426, -70.546]
  MoveL 124 to (730.32, 1092.57, 532.29) mm, rotated rx 180 ry 0 rz -88.32 deg; joints [46.452, -45.192, -61.46, 43.93, -49.371, -70.368]
  MoveL 125 to (727.64, 1093.52, 532.29) mm, rotated rx -180 ry 0 rz -88.32 deg; joints [46.31, -45.298, -61.514, 43.854, -49.314, -70.19]
  MoveL 126 to (724.95, 1094.47, 532.29) mm, rotated rx 180 ry 0 rz -88.32 deg; joints [46.168, -45.404, -61.566, 43.777, -49.258, -70.012]
  MoveL 127 to (722.27, 1095.43, 532.29) mm, rotated rx 180 ry 0 rz -88.32 deg; joints [46.024, -45.508, -61.618, 43.7, -49.2, -69.833]
  MoveL 128 to (719.59, 1096.4, 532.29) mm, rotated rx 180 ry 0 rz -88.32 deg; joints [45.881, -45.612, -61.67, 43.623, -49.143, -69.653]
  MoveL 129 to (716.91, 1097.37, 532.29) mm, rotated rx -180 ry 0 rz -88.32 deg; joints [45.737, -45.714, -61.721, 43.545, -49.085, -69.473]
  MoveL 130 to (714.24, 1098.36, 532.29) mm, rotated rx -180 ry 0 rz -88.32 deg; joints [45.592, -45.816, -61.771, 43.467, -49.026, -69.293]
  MoveL 131 to (711.56, 1099.35, 532.29) mm, rotated rx 180 ry 0 rz -88.32 deg; joints [45.447, -45.916, -61.821, 43.388, -48.967, -69.113]
  MoveL 132 to (708.89, 1100.35, 532.29) mm, rotated rx 180 ry 0 rz -88.32 deg; joints [45.301, -46.016, -61.87, 43.309, -48.907, -68.931]
  MoveL 133 to (706.23, 1101.35, 532.29) mm, rotated rx 180 ry 0 rz -88.32 deg; joints [45.154, -46.114, -61.919, 43.23, -48.847, -68.75]
  MoveL 134 to (703.56, 1102.37, 532.29) mm, rotated rx 180 ry 0 rz -88.32 deg; joints [45.008, -46.212, -61.967, 43.15, -48.786, -68.568]
  MoveL 135 to (700.9, 1103.39, 532.29) mm, rotated rx -180 ry 0 rz -88.32 deg; joints [44.86, -46.308, -62.014, 43.07, -48.725, -68.386]
  MoveL 136 to (698.25, 1104.42, 532.29) mm, rotated rx -180 ry 0 rz -88.32 deg; joints [44.712, -46.403, -62.061, 42.989, -48.663, -68.203]
  MoveL 137 to (695.59, 1105.45, 532.29) mm, rotated rx 180 ry 0 rz -88.32 deg; joints [44.564, -46.498, -62.108, 42.908, -48.601, -68.02]
  MoveL 138 to (692.94, 1106.5, 532.29) mm, rotated rx 180 ry 0 rz -88.32 deg; joints [44.415, -46.591, -62.153, 42.827, -48.538, -67.837]
  MoveL 139 to (690.29, 1107.55, 532.29) mm, rotated rx -180 ry 0 rz -88.32 deg; joints [44.265, -46.683, -62.198, 42.745, -48.475, -67.653]
  MoveL 140 to (687.64, 1108.61, 532.29) mm, rotated rx -180 ry 0 rz -88.32 deg; joints [44.115, -46.774, -62.243, 42.663, -48.411, -67.469]
  MoveL 141 to (685, 1109.67, 532.29) mm, rotated rx 180 ry 0 rz -88.32 deg; joints [43.965, -46.864, -62.287, 42.58, -48.347, -67.285]
  MoveL 142 to (682.36, 1110.75, 532.29) mm, rotated rx 180 ry 0 rz -88.32 deg; joints [43.814, -46.953, -62.33, 42.498, -48.282, -67.1]
  MoveL 143 to (679.72, 1111.83, 532.29) mm, rotated rx 180 ry 0 rz -88.32 deg; joints [43.663, -47.041, -62.373, 42.414, -48.217, -66.915]
  MoveL 144 to (677.09, 1112.91, 532.29) mm, rotated rx 180 ry 0 rz -88.32 deg; joints [43.511, -47.127, -62.415, 42.331, -48.151, -66.729]
  MoveL 145 to (674.46, 1114.01, 532.29) mm, rotated rx -180 ry 0 rz -88.32 deg; joints [43.358, -47.213, -62.456, 42.247, -48.084, -66.543]
  MoveL 146 to (671.83, 1115.11, 532.29) mm, rotated rx -180 ry 0 rz -88.32 deg; joints [43.206, -47.297, -62.497, 42.163, -48.018, -66.357]
  MoveL 147 to (669.21, 1116.22, 532.29) mm, rotated rx -180 ry 0 rz -88.32 deg; joints [43.052, -47.38, -62.537, 42.078, -47.95, -66.171]
  MoveL 148 to (666.58, 1117.34, 532.29) mm, rotated rx 180 ry 0 rz -88.32 deg; joints [42.899, -47.462, -62.577, 41.993, -47.882, -65.984]
  MoveL 149 to (663.97, 1118.46, 532.29) mm, rotated rx -180 ry 0 rz -88.32 deg; joints [42.744, -47.543, -62.616, 41.907, -47.814, -65.797]
  MoveL 150 to (661.35, 1119.6, 532.29) mm, rotated rx -180 ry 0 rz -88.32 deg; joints [42.59, -47.623, -62.654, 41.822, -47.745, -65.609]
  MoveL 151 to (658.74, 1120.74, 532.29) mm, rotated rx 180 ry 0 rz -88.32 deg; joints [42.435, -47.701, -62.692, 41.736, -47.676, -65.422]
  MoveL 152 to (656.13, 1121.88, 532.29) mm, rotated rx -180 ry 0 rz -88.32 deg; joints [42.279, -47.779, -62.729, 41.649, -47.606, -65.234]
  MoveL 153 to (653.52, 1123.04, 532.29) mm, rotated rx 180 ry 0 rz -88.32 deg; joints [42.123, -47.855, -62.766, 41.562, -47.535, -65.045]
  MoveL 154 to (650.92, 1124.2, 532.29) mm, rotated rx 180 ry 0 rz -88.32 deg; joints [41.967, -47.93, -62.802, 41.475, -47.464, -64.857]
  MoveL 155 to (648.32, 1125.37, 532.29) mm, rotated rx 180 ry 0 rz -88.32 deg; joints [41.81, -48.004, -62.837, 41.387, -47.393, -64.668]
  MoveL 156 to (645.73, 1126.54, 532.29) mm, rotated rx -180 ry 0 rz -88.32 deg; joints [41.653, -48.076, -62.872, 41.3, -47.321, -64.479]
  MoveL 157 to (643.13, 1127.73, 532.29) mm, rotated rx -180 ry 0 rz -88.32 deg; joints [41.495, -48.148, -62.906, 41.211, -47.248, -64.29]
  MoveL 158 to (640.54, 1128.92, 532.29) mm, rotated rx -180 ry 0 rz -88.32 deg; joints [41.337, -48.218, -62.94, 41.123, -47.175, -64.1]
  MoveL 159 to (637.96, 1130.11, 532.29) mm, rotated rx 180 ry 0 rz -88.32 deg; joints [41.179, -48.287, -62.972, 41.034, -47.102, -63.91]
  MoveL 160 to (635.38, 1131.32, 532.29) mm, rotated rx 180 ry 0 rz -88.32 deg; joints [41.02, -48.354, -63.005, 40.944, -47.028, -63.72]
  MoveL 161 to (632.8, 1132.53, 532.29) mm, rotated rx -180 ry 0 rz -88.32 deg; joints [40.861, -48.421, -63.036, 40.855, -46.953, -63.53]
  MoveL 162 to (630.22, 1133.75, 532.29) mm, rotated rx -180 ry 0 rz -88.32 deg; joints [40.701, -48.486, -63.067, 40.765, -46.878, -63.339]
  MoveL 163 to (627.65, 1134.98, 532.29) mm, rotated rx 180 ry 0 rz -88.32 deg; joints [40.541, -48.55, -63.097, 40.675, -46.803, -63.148]
  MoveL 164 to (625.08, 1136.21, 532.29) mm, rotated rx -180 ry 0 rz -88.32 deg; joints [40.381, -48.612, -63.127, 40.584, -46.727, -62.957]
  MoveL 165 to (622.51, 1137.45, 532.29) mm, rotated rx -180 ry 0 rz -88.32 deg; joints [40.22, -48.673, -63.156, 40.493, -46.65, -62.766]
  MoveL 166 to (619.95, 1138.7, 532.29) mm, rotated rx -180 ry 0 rz -88.32 deg; joints [40.059, -48.733, -63.185, 40.402, -46.573, -62.575]
  MoveL 167 to (617.39, 1139.96, 532.29) mm, rotated rx 180 ry 0 rz -88.32 deg; joints [39.898, -48.792, -63.212, 40.31, -46.495, -62.383]
  MoveL 168 to (614.84, 1141.22, 532.29) mm, rotated rx -180 ry 0 rz -88.32 deg; joints [39.737, -48.85, -63.24, 40.218, -46.417, -62.191]
  MoveL 169 to (612.29, 1142.49, 532.29) mm, rotated rx 180 ry 0 rz -88.32 deg; joints [39.575, -48.906, -63.266, 40.126, -46.339, -61.999]
  MoveL 170 to (609.74, 1143.77, 532.29) mm, rotated rx -180 ry 0 rz -88.32 deg; joints [39.412, -48.96, -63.292, 40.033, -46.26, -61.807]
  MoveL 171 to (607.2, 1145.05, 532.29) mm, rotated rx 180 ry 0 rz -88.32 deg; joints [39.25, -49.014, -63.317, 39.941, -46.18, -61.615]
  MoveL 172 to (604.66, 1146.34, 532.29) mm, rotated rx -180 ry 0 rz -88.32 deg; joints [39.087, -49.066, -63.342, 39.847, -46.1, -61.422]
  MoveL 173 to (602.12, 1147.64, 532.29) mm, rotated rx 180 ry 0 rz -88.32 deg; joints [38.924, -49.117, -63.366, 39.754, -46.02, -61.23]
  MoveL 174 to (599.58, 1148.95, 532.29) mm, rotated rx -180 ry 0 rz -88.32 deg; joints [38.76, -49.166, -63.389, 39.66, -45.938, -61.037]
  MoveL 175 to (597.06, 1150.26, 532.29) mm, rotated rx -180 ry 0 rz -88.32 deg; joints [38.596, -49.215, -63.411, 39.566, -45.857, -60.844]
  MoveL 176 to (594.53, 1151.58, 532.29) mm, rotated rx -180 ry 0 rz -88.32 deg; joints [38.432, -49.261, -63.433, 39.472, -45.775, -60.651]
  MoveL 177 to (592.01, 1152.9, 532.29) mm, rotated rx -180 ry 0 rz -88.32 deg; joints [38.268, -49.307, -63.455, 39.377, -45.692, -60.457]
  MoveL 178 to (589.49, 1154.24, 532.29) mm, rotated rx -180 ry 0 rz -88.32 deg; joints [38.104, -49.351, -63.475, 39.282, -45.609, -60.264]
  MoveL 179 to (586.97, 1155.58, 532.29) mm, rotated rx -180 ry 0 rz -88.32 deg; joints [37.939, -49.394, -63.495, 39.187, -45.526, -60.071]
  MoveL 180 to (584.46, 1156.93, 532.29) mm, rotated rx -180 ry 0 rz -88.32 deg; joints [37.774, -49.435, -63.515, 39.091, -45.442, -59.877]
  MoveL 181 to (581.96, 1158.28, 532.29) mm, rotated rx -180 ry 0 rz -88.32 deg; joints [37.608, -49.475, -63.534, 38.995, -45.358, -59.683]
  MoveL 182 to (579.45, 1159.64, 532.29) mm, rotated rx 180 ry 0 rz -88.32 deg; joints [37.443, -49.514, -63.552, 38.899, -45.273, -59.489]
  MoveL 183 to (576.95, 1161.01, 532.29) mm, rotated rx -180 ry 0 rz -88.32 deg; joints [37.277, -49.551, -63.569, 38.803, -45.187, -59.295]
  MoveL 184 to (574.46, 1162.39, 532.29) mm, rotated rx -180 ry 0 rz -88.32 deg; joints [37.111, -49.587, -63.586, 38.706, -45.101, -59.101]
  MoveL 185 to (571.97, 1163.77, 532.29) mm, rotated rx 180 ry 0 rz -88.32 deg; joints [36.945, -49.622, -63.602, 38.609, -45.015, -58.907]
  MoveL 186 to (569.48, 1165.16, 532.29) mm, rotated rx -180 ry 0 rz -88.32 deg; joints [36.779, -49.655, -63.617, 38.512, -44.928, -58.713]
  MoveL 187 to (566.99, 1166.56, 532.29) mm, rotated rx 180 ry 0 rz -88.32 deg; joints [36.612, -49.686, -63.632, 38.414, -44.841, -58.519]
  MoveL 188 to (564.51, 1167.96, 532.29) mm, rotated rx -180 ry 0 rz -88.32 deg; joints [36.446, -49.717, -63.646, 38.317, -44.753, -58.325]
  MoveL 189 to (562.04, 1169.37, 532.29) mm, rotated rx 180 ry 0 rz -88.32 deg; joints [36.279, -49.746, -63.66, 38.219, -44.665, -58.13]
  MoveL 190 to (559.57, 1170.79, 532.29) mm, rotated rx -180 ry 0 rz -88.32 deg; joints [36.112, -49.773, -63.673, 38.12, -44.576, -57.936]
  MoveL 191 to (557.1, 1172.22, 532.29) mm, rotated rx 180 ry 0 rz -88.32 deg; joints [35.944, -49.799, -63.685, 38.022, -44.487, -57.741]
  MoveL 192 to (554.63, 1173.65, 532.29) mm, rotated rx -180 ry 0 rz -88.32 deg; joints [35.777, -49.824, -63.696, 37.923, -44.398, -57.547]
  MoveL 193 to (552.17, 1175.09, 532.29) mm, rotated rx 180 ry 0 rz -88.32 deg; joints [35.61, -49.847, -63.707, 37.824, -44.308, -57.352]
  MoveL 194 to (549.72, 1176.53, 532.29) mm, rotated rx -180 ry 0 rz -88.32 deg; joints [35.442, -49.869, -63.717, 37.725, -44.217, -57.158]
  MoveL 195 to (547.27, 1177.99, 532.29) mm, rotated rx -180 ry 0 rz -88.32 deg; joints [35.274, -49.89, -63.727, 37.625, -44.126, -56.963]
  MoveL 196 to (544.82, 1179.44, 532.29) mm, rotated rx -180 ry 0 rz -88.32 deg; joints [35.106, -49.909, -63.736, 37.526, -44.035, -56.768]
  MoveL 197 to (542.37, 1180.91, 532.29) mm, rotated rx 180 ry 0 rz -88.32 deg; joints [34.938, -49.927, -63.744, 37.426, -43.943, -56.574]
  MoveL 198 to (539.93, 1182.38, 532.29) mm, rotated rx -180 ry 0 rz -88.32 deg; joints [34.77, -49.943, -63.751, 37.326, -43.851, -56.379]
  MoveL 199 to (537.5, 1183.86, 532.29) mm, rotated rx -180 ry 0 rz -88.32 deg; joints [34.602, -49.958, -63.758, 37.225, -43.759, -56.184]
  MoveL 200 to (535.07, 1185.35, 532.29) mm, rotated rx -180 ry 0 rz -88.32 deg; joints [34.434, -49.971, -63.765, 37.125, -43.666, -55.99]
  MoveL 201 to (532.64, 1186.84, 532.29) mm, rotated rx -180 ry 0 rz -88.32 deg; joints [34.266, -49.983, -63.77, 37.024, -43.572, -55.795]
  MoveL 202 to (530.22, 1188.34, 532.29) mm, rotated rx -180 ry 0 rz -88.32 deg; joints [34.097, -49.993, -63.775, 36.923, -43.478, -55.6]
  MoveL 203 to (527.8, 1189.85, 532.29) mm, rotated rx -180 ry 0 rz -88.32 deg; joints [33.929, -50.003, -63.779, 36.822, -43.384, -55.406]
  MoveL 204 to (525.38, 1191.36, 532.29) mm, rotated rx -180 ry 0 rz -88.32 deg; joints [33.76, -50.01, -63.783, 36.72, -43.289, -55.211]
  MoveL 205 to (522.97, 1192.88, 532.29) mm, rotated rx -180 ry 0 rz -88.32 deg; joints [33.592, -50.016, -63.786, 36.619, -43.194, -55.017]
  MoveL 206 to (520.57, 1194.41, 532.29) mm, rotated rx 180 ry 0 rz -88.32 deg; joints [33.423, -50.021, -63.788, 36.517, -43.099, -54.822]
  MoveL 207 to (518.17, 1195.95, 532.29) mm, rotated rx 180 ry 0 rz -88.32 deg; joints [33.255, -50.025, -63.789, 36.415, -43.003, -54.628]
  MoveL 208 to (515.77, 1197.49, 532.29) mm, rotated rx -180 ry 0 rz -88.32 deg; joints [33.086, -50.026, -63.79, 36.313, -42.907, -54.433]
  MoveL 209 to (513.37, 1199.03, 532.29) mm, rotated rx -180 ry 0 rz -88.32 deg; joints [32.917, -50.027, -63.791, 36.21, -42.81, -54.239]
  MoveL 210 to (510.99, 1200.59, 532.29) mm, rotated rx -180 ry 0 rz -88.32 deg; joints [32.749, -50.026, -63.79, 36.108, -42.713, -54.044]
  MoveL 211 to (508.6, 1202.15, 532.29) mm, rotated rx -180 ry 0 rz -88.32 deg; joints [32.58, -50.024, -63.789, 36.005, -42.616, -53.85]
  MoveL 212 to (506.22, 1203.72, 532.29) mm, rotated rx -180 ry 0 rz -88.32 deg; joints [32.411, -50.02, -63.787, 35.902, -42.518, -53.656]
  MoveL 213 to (503.85, 1205.29, 532.29) mm, rotated rx -180 ry 0 rz -88.32 deg; joints [32.243, -50.015, -63.785, 35.799, -42.42, -53.462]
  MoveL 214 to (501.47, 1206.87, 532.29) mm, rotated rx -180 ry 0 rz -88.32 deg; joints [32.074, -50.008, -63.782, 35.696, -42.321, -53.268]
  MoveL 215 to (499.11, 1208.46, 532.29) mm, rotated rx -180 ry 0 rz -88.32 deg; joints [31.906, -50, -63.778, 35.592, -42.222, -53.074]
  MoveL 216 to (496.75, 1210.05, 532.29) mm, rotated rx -180 ry 0 rz -88.32 deg; joints [31.737, -49.99, -63.773, 35.489, -42.123, -52.88]
  MoveL 217 to (494.39, 1211.65, 532.29) mm, rotated rx -180 ry 0 rz -88.32 deg; joints [31.569, -49.979, -63.768, 35.385, -42.023, -52.686]
  MoveL 218 to (492.03, 1213.26, 532.29) mm, rotated rx -180 ry 0 rz -88.32 deg; joints [31.401, -49.967, -63.763, 35.281, -41.923, -52.493]
  MoveL 219 to (489.69, 1214.88, 532.29) mm, rotated rx 180 ry 0 rz -88.32 deg; joints [31.233, -49.953, -63.756, 35.177, -41.823, -52.299]
  MoveL 220 to (487.34, 1216.5, 532.29) mm, rotated rx 180 ry 0 rz -88.32 deg; joints [31.064, -49.938, -63.749, 35.073, -41.722, -52.106]
  MoveL 221 to (485, 1218.12, 532.29) mm, rotated rx 180 ry 0 rz -88.32 deg; joints [30.896, -49.921, -63.741, 34.969, -41.622, -51.912]
  MoveL 222 to (482.67, 1219.76, 532.29) mm, rotated rx -180 ry 0 rz -88.32 deg; joints [30.728, -49.903, -63.733, 34.865, -41.52, -51.719]
  MoveL 223 to (480.34, 1221.4, 532.29) mm, rotated rx -180 ry 0 rz -88.32 deg; joints [30.561, -49.884, -63.724, 34.76, -41.419, -51.526]
  MoveL 224 to (478.01, 1223.04, 532.29) mm, rotated rx -180 ry 0 rz -88.32 deg; joints [30.393, -49.863, -63.714, 34.656, -41.317, -51.333]
  MoveL 225 to (475.69, 1224.7, 532.29) mm, rotated rx -180 ry 0 rz -88.32 deg; joints [30.225, -49.84, -63.704, 34.551, -41.214, -51.141]
  MoveL 226 to (473.37, 1226.36, 532.29) mm, rotated rx 180 ry 0 rz -88.32 deg; joints [30.058, -49.816, -63.693, 34.446, -41.112, -50.948]
  MoveL 227 to (471.06, 1228.02, 532.29) mm, rotated rx 180 ry 0 rz -88.32 deg; joints [29.891, -49.791, -63.681, 34.341, -41.009, -50.756]
  MoveL 228 to (468.75, 1229.7, 532.29) mm, rotated rx -180 ry 0 rz -88.32 deg; joints [29.723, -49.765, -63.669, 34.236, -40.906, -50.563]
  MoveL 229 to (466.45, 1231.38, 532.29) mm, rotated rx -180 ry 0 rz -88.32 deg; joints [29.556, -49.737, -63.656, 34.131, -40.802, -50.371]
  MoveL 230 to (464.15, 1233.06, 532.29) mm, rotated rx -180 ry 0 rz -88.32 deg; joints [29.39, -49.707, -63.642, 34.025, -40.699, -50.179]
  MoveL 231 to (461.86, 1234.75, 532.29) mm, rotated rx -180 ry 0 rz -88.32 deg; joints [29.223, -49.677, -63.628, 33.92, -40.595, -49.987]
  MoveL 232 to (459.57, 1236.45, 532.29) mm, rotated rx -180 ry 0 rz -88.32 deg; joints [29.056, -49.644, -63.613, 33.815, -40.49, -49.796]
  MoveL 233 to (457.29, 1238.16, 532.29) mm, rotated rx -180 ry 0 rz -88.32 deg; joints [28.89, -49.611, -63.597, 33.709, -40.386, -49.604]
  MoveL 234 to (455.01, 1239.87, 532.29) mm, rotated rx 180 ry 0 rz -88.32 deg; joints [28.724, -49.576, -63.581, 33.603, -40.281, -49.413]
  MoveL 235 to (452.74, 1241.59, 532.29) mm, rotated rx -180 ry 0 rz -88.32 deg; joints [28.558, -49.54, -63.564, 33.498, -40.176, -49.222]
  MoveL 236 to (450.47, 1243.31, 532.29) mm, rotated rx -180 ry 0 rz -88.32 deg; joints [28.393, -49.502, -63.546, 33.392, -40.071, -49.031]
  MoveL 237 to (448.2, 1245.04, 532.29) mm, rotated rx -180 ry 0 rz -88.32 deg; joints [28.227, -49.463, -63.528, 33.286, -39.965, -48.84]
  MoveL 238 to (445.94, 1246.78, 532.29) mm, rotated rx 180 ry 0 rz -88.32 deg; joints [28.062, -49.422, -63.509, 33.18, -39.859, -48.65]
  MoveL 239 to (443.69, 1248.52, 532.29) mm, rotated rx -180 ry 0 rz -88.32 deg; joints [27.897, -49.38, -63.489, 33.074, -39.753, -48.459]
  MoveL 240 to (441.44, 1250.27, 532.29) mm, rotated rx 180 ry 0 rz -88.32 deg; joints [27.732, -49.337, -63.469, 32.968, -39.647, -48.269]
  MoveL 241 to (439.19, 1252.03, 532.29) mm, rotated rx -180 ry 0 rz -88.32 deg; joints [27.568, -49.293, -63.448, 32.862, -39.54, -48.079]
  MoveL 242 to (436.95, 1253.79, 532.29) mm, rotated rx -180 ry 0 rz -88.32 deg; joints [27.404, -49.247, -63.427, 32.755, -39.434, -47.89]
  MoveL 243 to (434.72, 1255.56, 532.29) mm, rotated rx -180 ry 0 rz -88.32 deg; joints [27.24, -49.2, -63.404, 32.649, -39.327, -47.7]
  MoveL 244 to (432.49, 1257.33, 532.29) mm, rotated rx -180 ry 0 rz -88.32 deg; joints [27.076, -49.151, -63.382, 32.543, -39.219, -47.511]
  MoveL 245 to (430.26, 1259.11, 532.29) mm, rotated rx 180 ry 0 rz -88.32 deg; joints [26.913, -49.101, -63.358, 32.437, -39.112, -47.322]
  MoveL 246 to (428.04, 1260.9, 532.29) mm, rotated rx 180 ry 0 rz -88.32 deg; joints [26.749, -49.05, -63.334, 32.33, -39.004, -47.133]
  MoveL 247 to (425.83, 1262.69, 532.29) mm, rotated rx -180 ry 0 rz -88.32 deg; joints [26.587, -48.997, -63.309, 32.224, -38.897, -46.945]
  MoveL 248 to (423.62, 1264.49, 532.29) mm, rotated rx 180 ry 0 rz -88.32 deg; joints [26.424, -48.943, -63.284, 32.117, -38.789, -46.756]
  MoveL 249 to (421.41, 1266.3, 532.29) mm, rotated rx 180 ry 0 rz -88.32 deg; joints [26.262, -48.888, -63.258, 32.011, -38.681, -46.568]
  MoveL 250 to (419.21, 1268.11, 532.29) mm, rotated rx -180 ry 0 rz -88.32 deg; joints [26.1, -48.832, -63.231, 31.904, -38.572, -46.38]
  MoveL 251 to (417.02, 1269.93, 532.29) mm, rotated rx -180 ry 0 rz -88.32 deg; joints [25.939, -48.774, -63.204, 31.798, -38.464, -46.193]
  MoveL 252 to (414.83, 1271.75, 532.29) mm, rotated rx 180 ry 0 rz -88.32 deg; joints [25.777, -48.715, -63.176, 31.691, -38.355, -46.006]
  MoveL 253 to (412.65, 1273.58, 532.29) mm, rotated rx -180 ry 0 rz -88.32 deg; joints [25.617, -48.654, -63.147, 31.585, -38.247, -45.819]
  MoveL 254 to (410.47, 1275.42, 532.29) mm, rotated rx 180 ry 0 rz -88.32 deg; joints [25.456, -48.593, -63.118, 31.478, -38.138, -45.632]
  MoveL 255 to (408.29, 1277.26, 532.29) mm, rotated rx 180 ry 0 rz -88.32 deg; joints [25.296, -48.53, -63.088, 31.372, -38.029, -45.445]
  MoveL 256 to (406.12, 1279.11, 532.29) mm, rotated rx 180 ry 0 rz -88.32 deg; joints [25.136, -48.465, -63.057, 31.265, -37.919, -45.259]
  MoveL 257 to (403.96, 1280.97, 532.29) mm, rotated rx 180 ry 0 rz -88.32 deg; joints [24.977, -48.4, -63.026, 31.158, -37.81, -45.073]
  MoveL 258 to (401.8, 1282.83, 532.29) mm, rotated rx -180 ry 0 rz -88.32 deg; joints [24.818, -48.333, -62.995, 31.052, -37.701, -44.888]
  MoveL 259 to (399.65, 1284.69, 532.29) mm, rotated rx 180 ry 0 rz -88.32 deg; joints [24.659, -48.265, -62.962, 30.945, -37.591, -44.702]
  MoveL 260 to (397.5, 1286.57, 532.29) mm, rotated rx 180 ry 0 rz -88.32 deg; joints [24.501, -48.196, -62.929, 30.839, -37.481, -44.517]
  MoveL 261 to (395.36, 1288.44, 532.29) mm, rotated rx -180 ry 0 rz -88.32 deg; joints [24.343, -48.125, -62.895, 30.732, -37.372, -44.332]
  MoveL 262 to (393.22, 1290.33, 532.29) mm, rotated rx 180 ry 0 rz -88.32 deg; joints [24.185, -48.054, -62.861, 30.626, -37.262, -44.148]
  MoveL 263 to (391.09, 1292.22, 532.29) mm, rotated rx -180 ry 0 rz -88.32 deg; joints [24.028, -47.981, -62.826, 30.519, -37.152, -43.964]
  MoveL 264 to (388.96, 1294.12, 532.29) mm, rotated rx 180 ry 0 rz -88.32 deg; joints [23.872, -47.906, -62.791, 30.413, -37.042, -43.78]
  MoveL 265 to (386.84, 1296.02, 532.29) mm, rotated rx 180 ry 0 rz -88.32 deg; joints [23.715, -47.831, -62.755, 30.306, -36.932, -43.596]
  MoveL 266 to (384.72, 1297.93, 532.29) mm, rotated rx -180 ry 0 rz -88.32 deg; joints [23.56, -47.755, -62.718, 30.2, -36.821, -43.413]
  MoveL 267 to (382.61, 1299.84, 532.29) mm, rotated rx -180 ry 0 rz -88.32 deg; joints [23.404, -47.677, -62.68, 30.093, -36.711, -43.23]
  MoveL 268 to (380.51, 1301.76, 532.29) mm, rotated rx -180 ry 0 rz -88.32 deg; joints [23.249, -47.598, -62.642, 29.987, -36.601, -43.047]
  MoveL 269 to (378.41, 1303.69, 532.29) mm, rotated rx 180 ry 0 rz -88.32 deg; joints [23.095, -47.518, -62.604, 29.88, -36.49, -42.865]
  MoveL 270 to (376.31, 1305.62, 532.29) mm, rotated rx 180 ry 0 rz -88.32 deg; joints [22.941, -47.437, -62.565, 29.774, -36.38, -42.683]
  MoveL 271 to (374.22, 1307.56, 532.29) mm, rotated rx -180 ry 0 rz -88.32 deg; joints [22.787, -47.354, -62.525, 29.668, -36.269, -42.501]
  MoveL 272 to (372.14, 1309.51, 532.29) mm, rotated rx -180 ry 0 rz -88.32 deg; joints [22.634, -47.271, -62.484, 29.562, -36.159, -42.319]
  MoveL 273 to (370.06, 1311.46, 532.29) mm, rotated rx -180 ry 0 rz -88.32 deg; joints [22.481, -47.186, -62.443, 29.455, -36.048, -42.138]
  MoveL 274 to (367.99, 1313.41, 532.29) mm, rotated rx 180 ry 0 rz -88.32 deg; joints [22.329, -47.1, -62.401, 29.349, -35.938, -41.958]
  MoveL 275 to (365.92, 1315.37, 532.29) mm, rotated rx -180 ry 0 rz -88.32 deg; joints [22.177, -47.013, -62.359, 29.243, -35.827, -41.777]
  MoveL 276 to (363.86, 1317.34, 532.29) mm, rotated rx -180 ry 0 rz -88.32 deg; joints [22.026, -46.925, -62.316, 29.137, -35.716, -41.597]
  MoveL 277 to (361.8, 1319.31, 532.29) mm, rotated rx -180 ry 0 rz -88.32 deg; joints [21.875, -46.836, -62.273, 29.031, -35.606, -41.417]
  MoveL 278 to (359.75, 1321.29, 532.29) mm, rotated rx -180 ry 0 rz -88.32 deg; joints [21.725, -46.745, -62.229, 28.925, -35.495, -41.238]
  MoveL 279 to (357.71, 1323.28, 532.29) mm, rotated rx 180 ry 0 rz -88.32 deg; joints [21.575, -46.654, -62.184, 28.819, -35.385, -41.059]
  MoveL 280 to (355.67, 1325.27, 532.29) mm, rotated rx -180 ry 0 rz -88.32 deg; joints [21.426, -46.561, -62.139, 28.714, -35.274, -40.88]
  MoveL 281 to (353.63, 1327.26, 532.29) mm, rotated rx -180 ry 0 rz -88.32 deg; joints [21.277, -46.468, -62.093, 28.608, -35.163, -40.702]
  MoveL 282 to (351.6, 1329.27, 532.29) mm, rotated rx 180 ry 0 rz -88.32 deg; joints [21.129, -46.373, -62.047, 28.502, -35.053, -40.524]
  MoveL 283 to (349.58, 1331.27, 532.29) mm, rotated rx -180 ry 0 rz -88.32 deg; joints [20.981, -46.278, -61.999, 28.397, -34.942, -40.346]
  MoveL 284 to (347.56, 1333.29, 532.29) mm, rotated rx -180 ry 0 rz -88.32 deg; joints [20.834, -46.181, -61.952, 28.291, -34.832, -40.169]
  MoveL 285 to (345.55, 1335.3, 532.29) mm, rotated rx -180 ry 0 rz -88.32 deg; joints [20.687, -46.083, -61.904, 28.186, -34.721, -39.992]
  MoveL 286 to (343.55, 1337.33, 532.29) mm, rotated rx -180 ry 0 rz -88.32 deg; joints [20.541, -45.984, -61.855, 28.081, -34.611, -39.815]
  MoveL 287 to (341.55, 1339.36, 532.29) mm, rotated rx 180 ry 0 rz -88.32 deg; joints [20.395, -45.884, -61.805, 27.975, -34.501, -39.639]
  MoveL 288 to (339.55, 1341.39, 532.29) mm, rotated rx -180 ry 0 rz -88.32 deg; joints [20.25, -45.784, -61.755, 27.87, -34.39, -39.463]
  MoveL 289 to (337.56, 1343.44, 532.29) mm, rotated rx -180 ry 0 rz -88.32 deg; joints [20.106, -45.682, -61.705, 27.765, -34.28, -39.288]
  MoveL 290 to (335.58, 1345.48, 532.29) mm, rotated rx 180 ry 0 rz -88.32 deg; joints [19.962, -45.579, -61.654, 27.66, -34.17, -39.113]
  MoveL 291 to (333.6, 1347.54, 532.29) mm, rotated rx 180 ry 0 rz -88.32 deg; joints [19.818, -45.475, -61.602, 27.555, -34.06, -38.938]
  MoveL 292 to (331.63, 1349.59, 532.29) mm, rotated rx 180 ry 0 rz -88.32 deg; joints [19.675, -45.37, -61.55, 27.45, -33.95, -38.763]
  MoveL 293 to (329.67, 1351.66, 532.29) mm, rotated rx -180 ry 0 rz -88.32 deg; joints [19.533, -45.265, -61.497, 27.346, -33.84, -38.589]
  MoveL 294 to (327.71, 1353.73, 532.29) mm, rotated rx -180 ry 0 rz -88.32 deg; joints [19.391, -45.158, -61.444, 27.241, -33.73, -38.416]
  MoveL 295 to (325.75, 1355.8, 532.29) mm, rotated rx -180 ry 0 rz -88.32 deg; joints [19.25, -45.05, -61.39, 27.137, -33.621, -38.243]
  MoveL 296 to (323.8, 1357.88, 532.29) mm, rotated rx -180 ry 0 rz -88.32 deg; joints [19.109, -44.942, -61.335, 27.032, -33.511, -38.07]
  MoveL 297 to (321.86, 1359.96, 532.29) mm, rotated rx -180 ry 0 rz -88.32 deg; joints [18.969, -44.832, -61.28, 26.928, -33.402, -37.897]
  MoveL 298 to (319.92, 1362.06, 532.29) mm, rotated rx -180 ry 0 rz -88.32 deg; joints [18.829, -44.722, -61.224, 26.824, -33.292, -37.725]
  MoveL 299 to (317.99, 1364.15, 532.29) mm, rotated rx -180 ry 0 rz -88.32 deg; joints [18.69, -44.61, -61.168, 26.72, -33.183, -37.553]
  MoveL 300 to (316.07, 1366.25, 532.29) mm, rotated rx -180 ry 0 rz -88.32 deg; joints [18.552, -44.498, -61.111, 26.616, -33.074, -37.382]
  MoveL 301 to (314.15, 1368.36, 532.29) mm, rotated rx -180 ry 0 rz -88.32 deg; joints [18.414, -44.385, -61.054, 26.512, -32.965, -37.211]
  MoveL 302 to (312.24, 1370.47, 532.29) mm, rotated rx -180 ry 0 rz -88.32 deg; joints [18.277, -44.271, -60.996, 26.408, -32.856, -37.041]
  MoveL 303 to (310.33, 1372.59, 532.29) mm, rotated rx 180 ry 0 rz -88.32 deg; joints [18.141, -44.156, -60.937, 26.305, -32.748, -36.871]
  MoveL 304 to (308.43, 1374.71, 532.29) mm, rotated rx 180 ry 0 rz -88.32 deg; joints [18.005, -44.04, -60.878, 26.201, -32.639, -36.701]
  MoveL 305 to (306.53, 1376.84, 532.29) mm, rotated rx -180 ry 0 rz -88.32 deg; joints [17.869, -43.924, -60.819, 26.098, -32.531, -36.532]
  MoveL 306 to (304.64, 1378.98, 532.29) mm, rotated rx 180 ry 0 rz -88.32 deg; joints [17.734, -43.806, -60.759, 25.995, -32.423, -36.363]
  MoveL 307 to (302.76, 1381.11, 532.29) mm, rotated rx -180 ry 0 rz -88.32 deg; joints [17.6, -43.688, -60.698, 25.892, -32.315, -36.194]
  MoveL 308 to (300.88, 1383.26, 532.29) mm, rotated rx -180 ry 0 rz -88.32 deg; joints [17.466, -43.569, -60.637, 25.789, -32.207, -36.026]
  MoveL 309 to (299.01, 1385.41, 532.29) mm, rotated rx -180 ry 0 rz -88.32 deg; joints [17.333, -43.449, -60.575, 25.686, -32.099, -35.859]
  MoveL 310 to (297.15, 1387.56, 532.29) mm, rotated rx -180 ry 0 rz -88.32 deg; joints [17.201, -43.328, -60.513, 25.583, -31.992, -35.691]
  MoveL 311 to (295.29, 1389.72, 532.29) mm, rotated rx 180 ry 0 rz -88.32 deg; joints [17.069, -43.206, -60.45, 25.48, -31.884, -35.525]
  MoveL 312 to (293.44, 1391.89, 532.29) mm, rotated rx -180 ry 0 rz -88.32 deg; joints [16.938, -43.084, -60.387, 25.378, -31.777, -35.358]
  MoveL 313 to (291.59, 1394.06, 532.29) mm, rotated rx 180 ry 0 rz -88.32 deg; joints [16.808, -42.961, -60.323, 25.276, -31.67, -35.192]
  MoveL 314 to (289.75, 1396.23, 532.29) mm, rotated rx -180 ry 0 rz -88.32 deg; joints [16.678, -42.837, -60.259, 25.174, -31.564, -35.027]
  MoveL 315 to (287.91, 1398.41, 532.29) mm, rotated rx -180 ry 0 rz -88.32 deg; joints [16.548, -42.712, -60.194, 25.072, -31.457, -34.861]
  MoveL 316 to (286.08, 1400.6, 532.29) mm, rotated rx 180 ry 0 rz -88.32 deg; joints [16.42, -42.587, -60.129, 24.97, -31.351, -34.697]
  MoveL 317 to (284.26, 1402.79, 532.29) mm, rotated rx 180 ry 0 rz -88.32 deg; joints [16.292, -42.461, -60.063, 24.868, -31.245, -34.532]
  MoveL 318 to (282.45, 1404.99, 532.29) mm, rotated rx -180 ry 0 rz -88.32 deg; joints [16.164, -42.334, -59.996, 24.766, -31.139, -34.369]
  MoveL 319 to (280.64, 1407.19, 532.29) mm, rotated rx 180 ry 0 rz -88.32 deg; joints [16.037, -42.206, -59.929, 24.665, -31.033, -34.205]
  MoveL 320 to (278.83, 1409.4, 532.29) mm, rotated rx -180 ry 0 rz -88.32 deg; joints [15.911, -42.078, -59.862, 24.564, -30.928, -34.042]
  MoveL 321 to (277.03, 1411.61, 532.29) mm, rotated rx 180 ry 0 rz -88.32 deg; joints [15.786, -41.949, -59.794, 24.462, -30.823, -33.88]
  MoveL 322 to (275.24, 1413.82, 532.29) mm, rotated rx -180 ry 0 rz -88.32 deg; joints [15.661, -41.819, -59.725, 24.362, -30.718, -33.717]
  MoveL 323 to (273.46, 1416.04, 532.29) mm, rotated rx 180 ry 0 rz -88.32 deg; joints [15.536, -41.689, -59.656, 24.261, -30.613, -33.556]
  MoveL 324 to (271.68, 1418.27, 532.29) mm, rotated rx -180 ry 0 rz -88.32 deg; joints [15.413, -41.558, -59.587, 24.16, -30.509, -33.394]
  MoveL 325 to (269.91, 1420.5, 532.29) mm, rotated rx -180 ry 0 rz -88.32 deg; joints [15.29, -41.426, -59.517, 24.06, -30.405, -33.234]
  MoveL 326 to (268.14, 1422.74, 532.29) mm, rotated rx -180 ry 0 rz -88.32 deg; joints [15.167, -41.294, -59.446, 23.959, -30.301, -33.073]
  MoveL 327 to (266.38, 1424.98, 532.29) mm, rotated rx 180 ry 0 rz -88.32 deg; joints [15.046, -41.161, -59.375, 23.859, -30.197, -32.913]
  MoveL 328 to (264.62, 1427.23, 532.29) mm, rotated rx 180 ry 0 rz -88.32 deg; joints [14.925, -41.027, -59.304, 23.759, -30.094, -32.754]
  MoveL 329 to (262.88, 1429.48, 532.29) mm, rotated rx -180 ry 0 rz -88.32 deg; joints [14.804, -40.893, -59.232, 23.659, -29.991, -32.595]
  MoveL 330 to (261.14, 1431.73, 532.29) mm, rotated rx -180 ry 0 rz -88.32 deg; joints [14.684, -40.758, -59.159, 23.559, -29.888, -32.436]
  MoveL 331 to (259.4, 1433.99, 532.29) mm, rotated rx 180 ry 0 rz -88.32 deg; joints [14.565, -40.622, -59.086, 23.46, -29.786, -32.278]
  MoveL 332 to (257.67, 1436.26, 532.29) mm, rotated rx -180 ry 0 rz -88.32 deg; joints [14.447, -40.486, -59.013, 23.361, -29.684, -32.12]
  MoveL 333 to (255.95, 1438.53, 532.29) mm, rotated rx -180 ry 0 rz -88.32 deg; joints [14.329, -40.349, -58.939, 23.261, -29.582, -31.963]
  MoveL 334 to (254.23, 1440.8, 532.29) mm, rotated rx -180 ry 0 rz -88.32 deg; joints [14.212, -40.212, -58.864, 23.162, -29.48, -31.806]
  MoveL 335 to (252.52, 1443.08, 532.29) mm, rotated rx -180 ry 0 rz -88.32 deg; joints [14.095, -40.074, -58.79, 23.064, -29.379, -31.65]
  MoveL 336 to (250.82, 1445.37, 532.29) mm, rotated rx -180 ry 0 rz -88.32 deg; joints [13.979, -39.936, -58.714, 22.965, -29.278, -31.494]
  MoveL 337 to (249.12, 1447.66, 532.29) mm, rotated rx 180 ry 0 rz -88.32 deg; joints [13.864, -39.796, -58.638, 22.866, -29.177, -31.338]
  MoveL 338 to (247.43, 1449.95, 532.29) mm, rotated rx 180 ry 0 rz -88.32 deg; joints [13.749, -39.657, -58.562, 22.768, -29.077, -31.184]
  MoveL 339 to (245.75, 1452.25, 532.29) mm, rotated rx -180 ry 0 rz -88.32 deg; joints [13.635, -39.517, -58.485, 22.67, -28.977, -31.029]
  MoveL 340 to (244.07, 1454.56, 532.29) mm, rotated rx -180 ry 0 rz -88.32 deg; joints [13.522, -39.376, -58.408, 22.572, -28.877, -30.875]
  MoveL 341 to (242.4, 1456.87, 532.29) mm, rotated rx 180 ry 0 rz -88.32 deg; joints [13.409, -39.235, -58.33, 22.474, -28.777, -30.721]
  MoveL 342 to (240.74, 1459.18, 532.29) mm, rotated rx 180 ry 0 rz -88.32 deg; joints [13.297, -39.093, -58.252, 22.377, -28.678, -30.568]
  MoveL 343 to (239.08, 1461.5, 532.29) mm, rotated rx -180 ry 0 rz -88.32 deg; joints [13.186, -38.951, -58.173, 22.279, -28.58, -30.416]
  MoveL 344 to (237.43, 1463.82, 532.29) mm, rotated rx 180 ry 0 rz -88.32 deg; joints [13.075, -38.808, -58.094, 22.182, -28.481, -30.264]
  MoveL 345 to (235.78, 1466.15, 532.29) mm, rotated rx -180 ry 0 rz -88.32 deg; joints [12.965, -38.665, -58.015, 22.085, -28.383, -30.112]
  MoveL 346 to (234.14, 1468.48, 532.29) mm, rotated rx 180 ry 0 rz -88.32 deg; joints [12.856, -38.521, -57.935, 21.989, -28.285, -29.961]
  MoveL 347 to (232.51, 1470.81, 532.29) mm, rotated rx 180 ry 0 rz -88.32 deg; joints [12.747, -38.377, -57.854, 21.892, -28.188, -29.81]
  MoveL 348 to (230.89, 1473.16, 532.29) mm, rotated rx -180 ry 0 rz -88.32 deg; joints [12.639, -38.232, -57.773, 21.796, -28.091, -29.66]
  MoveL 349 to (229.27, 1475.5, 532.29) mm, rotated rx -180 ry 0 rz -88.32 deg; joints [12.531, -38.087, -57.692, 21.699, -27.994, -29.51]
  MoveL 350 to (227.66, 1477.85, 532.29) mm, rotated rx -180 ry 0 rz -88.32 deg; joints [12.425, -37.942, -57.61, 21.603, -27.898, -29.361]
  MoveL 351 to (226.05, 1480.21, 532.29) mm, rotated rx -180 ry 0 rz -88.32 deg; joints [12.319, -37.795, -57.528, 21.508, -27.802, -29.212]
  MoveL 352 to (224.45, 1482.57, 532.29) mm, rotated rx -180 ry 0 rz -88.32 deg; joints [12.213, -37.649, -57.445, 21.412, -27.706, -29.064]
  MoveL 353 to (222.86, 1484.93, 532.29) mm, rotated rx 180 ry 0 rz -88.32 deg; joints [12.108, -37.502, -57.362, 21.317, -27.611, -28.916]
  MoveL 354 to (221.27, 1487.3, 532.29) mm, rotated rx -180 ry 0 rz -88.32 deg; joints [12.004, -37.355, -57.278, 21.221, -27.516, -28.768]
  MoveL 355 to (219.69, 1489.67, 532.29) mm, rotated rx -180 ry 0 rz -88.32 deg; joints [11.901, -37.207, -57.194, 21.126, -27.421, -28.621]
  MoveL 356 to (218.12, 1492.05, 532.29) mm, rotated rx 180 ry 0 rz -88.32 deg; joints [11.798, -37.059, -57.11, 21.032, -27.327, -28.475]
  MoveL 357 to (216.56, 1494.43, 532.29) mm, rotated rx -180 ry 0 rz -88.32 deg; joints [11.695, -36.91, -57.025, 20.937, -27.233, -28.329]
  MoveL 358 to (215, 1496.81, 532.29) mm, rotated rx -180 ry 0 rz -88.32 deg; joints [11.594, -36.762, -56.94, 20.843, -27.14, -28.184]
  MoveL 359 to (213.45, 1499.2, 532.29) mm, rotated rx -180 ry 0 rz -88.32 deg; joints [11.493, -36.612, -56.854, 20.749, -27.047, -28.039]
  MoveL 360 to (211.9, 1501.6, 532.29) mm, rotated rx 180 ry 0 rz -88.32 deg; joints [11.393, -36.463, -56.768, 20.655, -26.954, -27.895]
  MoveL 361 to (210.36, 1504, 532.29) mm, rotated rx -180 ry 0 rz -88.32 deg; joints [11.293, -36.313, -56.681, 20.561, -26.862, -27.751]
  MoveL 362 to (208.83, 1506.4, 532.29) mm, rotated rx 180 ry 0 rz -88.32 deg; joints [11.194, -36.162, -56.594, 20.468, -26.77, -27.607]
  MoveL 363 to (207.3, 1508.81, 532.29) mm, rotated rx -180 ry 0 rz -88.32 deg; joints [11.096, -36.011, -56.507, 20.374, -26.678, -27.464]
  MoveL 364 to (205.78, 1511.22, 532.29) mm, rotated rx 180 ry 0 rz -88.32 deg; joints [10.998, -35.86, -56.419, 20.281, -26.587, -27.322]
  MoveL 365 to (204.27, 1513.63, 532.29) mm, rotated rx 180 ry 0 rz -88.32 deg; joints [10.901, -35.709, -56.331, 20.189, -26.497, -27.18]
  MoveL 366 to (202.77, 1516.05, 532.29) mm, rotated rx 180 ry 0 rz -88.32 deg; joints [10.804, -35.557, -56.242, 20.096, -26.406, -27.039]
  MoveL 367 to (201.27, 1518.48, 532.29) mm, rotated rx -180 ry 0 rz -88.32 deg; joints [10.709, -35.405, -56.153, 20.004, -26.316, -26.898]
  MoveL 368 to (199.78, 1520.91, 532.29) mm, rotated rx 180 ry 0 rz -88.32 deg; joints [10.614, -35.253, -56.063, 19.912, -26.227, -26.758]
  MoveL 369 to (198.29, 1523.34, 532.29) mm, rotated rx 180 ry 0 rz -88.32 deg; joints [10.519, -35.1, -55.974, 19.82, -26.138, -26.618]
  MoveL 370 to (196.82, 1525.78, 532.29) mm, rotated rx 180 ry 0 rz -88.32 deg; joints [10.425, -34.947, -55.883, 19.728, -26.049, -26.479]
  MoveL 371 to (195.34, 1528.22, 532.29) mm, rotated rx 180 ry 0 rz -88.32 deg; joints [10.332, -34.794, -55.793, 19.637, -25.961, -26.34]
  MoveL 372 to (193.88, 1530.66, 532.29) mm, rotated rx 180 ry 0 rz -88.32 deg; joints [10.24, -34.64, -55.702, 19.546, -25.873, -26.202]
  MoveL 373 to (192.42, 1533.11, 532.29) mm, rotated rx -180 ry 0 rz -88.32 deg; joints [10.148, -34.486, -55.61, 19.455, -25.785, -26.064]
  MoveL 374 to (190.97, 1535.56, 532.29) mm, rotated rx 180 ry 0 rz -88.32 deg; joints [10.056, -34.332, -55.518, 19.364, -25.698, -25.927]
  MoveL 375 to (189.53, 1538.02, 532.29) mm, rotated rx -180 ry 0 rz -88.32 deg; joints [9.966, -34.177, -55.426, 19.274, -25.612, -25.79]
  MoveL 376 to (188.09, 1540.48, 532.29) mm, rotated rx 180 ry 0 rz -88.32 deg; joints [9.876, -34.023, -55.333, 19.184, -25.525, -25.654]
  MoveL 377 to (186.66, 1542.95, 532.29) mm, rotated rx 180 ry 0 rz -88.32 deg; joints [9.786, -33.868, -55.24, 19.094, -25.44, -25.518]
  MoveL 378 to (185.24, 1545.42, 532.29) mm, rotated rx -180 ry 0 rz -88.32 deg; joints [9.697, -33.713, -55.147, 19.004, -25.354, -25.383]
  MoveL 379 to (183.82, 1547.89, 532.29) mm, rotated rx -180 ry 0 rz -88.32 deg; joints [9.609, -33.557, -55.053, 18.915, -25.269, -25.249]
  MoveL 380 to (182.41, 1550.37, 532.29) mm, rotated rx 180 ry 0 rz -88.32 deg; joints [9.522, -33.401, -54.959, 18.826, -25.185, -25.115]
  MoveL 381 to (181.01, 1552.85, 532.29) mm, rotated rx -180 ry 0 rz -88.32 deg; joints [9.435, -33.246, -54.864, 18.737, -25.101, -24.981]
  MoveL 382 to (179.62, 1555.33, 532.29) mm, rotated rx 180 ry 0 rz -88.32 deg; joints [9.349, -33.089, -54.77, 18.648, -25.017, -24.848]
  MoveL 383 to (178.23, 1557.82, 532.29) mm, rotated rx -180 ry 0 rz -88.32 deg; joints [9.263, -32.933, -54.674, 18.56, -24.934, -24.716]
  MoveL 384 to (176.85, 1560.31, 532.29) mm, rotated rx 180 ry 0 rz -88.32 deg; joints [9.178, -32.776, -54.579, 18.472, -24.851, -24.584]
  MoveL 385 to (175.47, 1562.81, 532.29) mm, rotated rx 180 ry 0 rz -88.32 deg; joints [9.094, -32.62, -54.483, 18.384, -24.768, -24.453]
  MoveL 386 to (174.11, 1565.31, 532.29) mm, rotated rx 180 ry 0 rz -88.32 deg; joints [9.01, -32.463, -54.386, 18.296, -24.687, -24.322]
  MoveL 387 to (172.75, 1567.82, 532.29) mm, rotated rx 180 ry 0 rz -88.32 deg; joints [8.927, -32.306, -54.289, 18.209, -24.605, -24.192]
  MoveL 388 to (171.39, 1570.32, 532.29) mm, rotated rx -180 ry 0 rz -88.32 deg; joints [8.844, -32.148, -54.192, 18.122, -24.524, -24.062]
  MoveL 389 to (170.05, 1572.84, 532.29) mm, rotated rx 180 ry 0 rz -88.32 deg; joints [8.763, -31.991, -54.095, 18.035, -24.443, -23.933]
  MoveL 390 to (168.71, 1575.35, 532.29) mm, rotated rx -180 ry 0 rz -88.32 deg; joints [8.681, -31.833, -53.997, 17.949, -24.363, -23.804]
  MoveL 391 to (167.38, 1577.87, 532.29) mm, rotated rx -180 ry 0 rz -88.32 deg; joints [8.601, -31.675, -53.899, 17.863, -24.283, -23.676]
  MoveL 392 to (166.05, 1580.4, 532.29) mm, rotated rx -180 ry 0 rz -88.32 deg; joints [8.521, -31.517, -53.8, 17.777, -24.204, -23.549]
  MoveL 393 to (164.74, 1582.92, 532.29) mm, rotated rx -180 ry 0 rz -88.32 deg; joints [8.441, -31.359, -53.701, 17.691, -24.125, -23.422]
  MoveL 394 to (163.43, 1585.45, 532.29) mm, rotated rx -180 ry 0 rz -88.32 deg; joints [8.362, -31.2, -53.602, 17.606, -24.047, -23.296]
  MoveL 395 to (162.12, 1587.99, 532.29) mm, rotated rx 180 ry 0 rz -88.32 deg; joints [8.284, -31.042, -53.502, 17.521, -23.969, -23.17]
  MoveL 396 to (160.83, 1590.53, 532.29) mm, rotated rx 180 ry 0 rz -88.32 deg; joints [8.206, -30.883, -53.402, 17.436, -23.891, -23.045]
  MoveL 397 to (159.54, 1593.07, 532.29) mm, rotated rx -180 ry 0 rz -88.32 deg; joints [8.129, -30.724, -53.302, 17.352, -23.814, -22.92]
  MoveL 398 to (158.25, 1595.61, 532.29) mm, rotated rx 180 ry 0 rz -88.32 deg; joints [8.053, -30.565, -53.201, 17.268, -23.737, -22.796]
  MoveL 399 to (156.98, 1598.16, 532.29) mm, rotated rx 180 ry 0 rz -88.32 deg; joints [7.977, -30.406, -53.101, 17.184, -23.661, -22.673]
  MoveL 400 to (155.71, 1600.71, 532.29) mm, rotated rx 180 ry 0 rz -88.32 deg; joints [7.902, -30.247, -52.999, 17.101, -23.585, -22.55]
  MoveL 401 to (154.45, 1603.27, 532.29) mm, rotated rx 180 ry 0 rz -88.32 deg; joints [7.827, -30.088, -52.898, 17.017, -23.51, -22.428]
  MoveL 402 to (153.2, 1605.83, 532.29) mm, rotated rx 180 ry 0 rz -88.32 deg; joints [7.753, -29.928, -52.796, 16.935, -23.435, -22.306]
  MoveL 403 to (151.95, 1608.39, 532.29) mm, rotated rx -180 ry 0 rz -88.32 deg; joints [7.68, -29.769, -52.693, 16.852, -23.361, -22.185]
  MoveL 404 to (150.71, 1610.96, 532.29) mm, rotated rx 180 ry 0 rz -88.32 deg; joints [7.607, -29.609, -52.591, 16.77, -23.287, -22.065]
  MoveL 405 to (149.48, 1613.53, 532.29) mm, rotated rx 180 ry 0 rz -88.32 deg; joints [7.535, -29.449, -52.488, 16.688, -23.213, -21.945]
  MoveL 406 to (148.26, 1616.1, 532.29) mm, rotated rx 180 ry 0 rz -88.32 deg; joints [7.463, -29.289, -52.384, 16.606, -23.14, -21.825]
  MoveL 407 to (147.04, 1618.68, 532.29) mm, rotated rx 180 ry 0 rz -88.32 deg; joints [7.392, -29.129, -52.281, 16.525, -23.067, -21.706]
  MoveL 408 to (145.83, 1621.26, 532.29) mm, rotated rx 180 ry 0 rz -88.32 deg; joints [7.322, -28.969, -52.177, 16.444, -22.995, -21.588]
  MoveL 409 to (144.62, 1623.84, 532.29) mm, rotated rx 180 ry 0 rz -88.32 deg; joints [7.252, -28.809, -52.072, 16.363, -22.924, -21.471]
  MoveL 410 to (143.43, 1626.43, 532.29) mm, rotated rx -180 ry 0 rz -88.32 deg; joints [7.182, -28.649, -51.968, 16.283, -22.852, -21.354]
  MoveL 411 to (142.24, 1629.02, 532.29) mm, rotated rx 180 ry 0 rz -88.32 deg; joints [7.114, -28.489, -51.863, 16.203, -22.782, -21.237]
  MoveL 412 to (141.06, 1631.61, 532.29) mm, rotated rx -180 ry 0 rz -88.32 deg; joints [7.045, -28.328, -51.758, 16.123, -22.711, -21.122]
  MoveL 413 to (139.89, 1634.21, 532.29) mm, rotated rx -180 ry 0 rz -88.32 deg; joints [6.978, -28.168, -51.652, 16.044, -22.641, -21.007]
  MoveL 414 to (138.72, 1636.81, 532.29) mm, rotated rx 180 ry 0 rz -88.32 deg; joints [6.911, -28.007, -51.546, 15.965, -22.572, -20.892]
  MoveL 415 to (137.56, 1639.41, 532.29) mm, rotated rx 180 ry 0 rz -88.32 deg; joints [6.844, -27.847, -51.44, 15.886, -22.503, -20.778]
  MoveL 416 to (136.41, 1642.02, 532.29) mm, rotated rx 180 ry 0 rz -88.32 deg; joints [6.778, -27.686, -51.334, 15.808, -22.434, -20.665]
  MoveL 417 to (135.26, 1644.63, 532.29) mm, rotated rx -180 ry 0 rz -88.32 deg; joints [6.713, -27.526, -51.227, 15.73, -22.366, -20.552]
  MoveL 418 to (134.13, 1647.24, 532.29) mm, rotated rx -180 ry 0 rz -88.32 deg; joints [6.648, -27.365, -51.12, 15.652, -22.299, -20.44]
  MoveL 419 to (133, 1649.86, 532.29) mm, rotated rx -180 ry 0 rz -88.32 deg; joints [6.584, -27.204, -51.012, 15.575, -22.231, -20.329]
  MoveL 420 to (131.87, 1652.48, 532.29) mm, rotated rx 180 ry 0 rz -88.32 deg; joints [6.521, -27.043, -50.905, 15.498, -22.165, -20.218]
  MoveL 421 to (130.76, 1655.1, 532.29) mm, rotated rx -180 ry 0 rz -88.32 deg; joints [6.457, -26.883, -50.797, 15.422, -22.098, -20.108]
  MoveL 422 to (129.65, 1657.73, 532.29) mm, rotated rx -180 ry 0 rz -88.32 deg; joints [6.395, -26.722, -50.688, 15.346, -22.033, -19.998]
  MoveL 423 to (128.55, 1660.35, 532.29) mm, rotated rx 180 ry 0 rz -88.32 deg; joints [6.333, -26.561, -50.58, 15.27, -21.967, -19.889]
  MoveL 424 to (127.46, 1662.99, 532.29) mm, rotated rx 180 ry 0 rz -88.32 deg; joints [6.272, -26.4, -50.471, 15.194, -21.902, -19.781]
  MoveL 425 to (126.37, 1665.62, 532.29) mm, rotated rx -180 ry 0 rz -88.32 deg; joints [6.211, -26.239, -50.362, 15.119, -21.838, -19.673]
  MoveL 426 to (125.29, 1668.26, 532.29) mm, rotated rx 180 ry 0 rz -88.32 deg; joints [6.15, -26.078, -50.252, 15.045, -21.774, -19.566]
  MoveL 427 to (124.22, 1670.9, 532.29) mm, rotated rx 180 ry 0 rz -88.32 deg; joints [6.091, -25.917, -50.142, 14.97, -21.71, -19.46]
  MoveL 428 to (123.16, 1673.54, 532.29) mm, rotated rx 180 ry 0 rz -88.32 deg; joints [6.031, -25.756, -50.032, 14.896, -21.647, -19.354]
  MoveL 429 to (122.1, 1676.19, 532.29) mm, rotated rx -180 ry 0 rz -88.32 deg; joints [5.973, -25.595, -49.922, 14.823, -21.585, -19.249]
  MoveL 430 to (121.05, 1678.84, 532.29) mm, rotated rx -180 ry 0 rz -88.32 deg; joints [5.915, -25.435, -49.811, 14.75, -21.523, -19.145]
  MoveL 431 to (120.01, 1681.49, 532.29) mm, rotated rx -180 ry 0 rz -88.32 deg; joints [5.857, -25.274, -49.7, 14.677, -21.461, -19.041]
  MoveL 432 to (118.98, 1684.15, 532.29) mm, rotated rx -180 ry 0 rz -88.32 deg; joints [5.8, -25.113, -49.589, 14.604, -21.4, -18.938]
  MoveL 433 to (117.95, 1686.81, 532.29) mm, rotated rx -180 ry 0 rz -88.32 deg; joints [5.743, -24.952, -49.478, 14.532, -21.339, -18.835]
  MoveL 434 to (116.93, 1689.47, 532.29) mm, rotated rx -180 ry 0 rz -88.32 deg; joints [5.687, -24.791, -49.366, 14.461, -21.278, -18.733]
  MoveL 435 to (115.92, 1692.13, 532.29) mm, rotated rx -180 ry 0 rz -88.32 deg; joints [5.632, -24.63, -49.254, 14.39, -21.218, -18.632]
  MoveL 436 to (114.91, 1694.8, 532.29) mm, rotated rx 180 ry 0 rz -88.32 deg; joints [5.577, -24.469, -49.142, 14.319, -21.159, -18.532]
  MoveL 437 to (113.92, 1697.47, 532.29) mm, rotated rx -180 ry 0 rz -88.32 deg; joints [5.522, -24.308, -49.029, 14.248, -21.1, -18.432]
  MoveL 438 to (112.93, 1700.14, 532.29) mm, rotated rx 180 ry 0 rz -88.32 deg; joints [5.469, -24.147, -48.916, 14.178, -21.041, -18.332]
  MoveL 439 to (111.95, 1702.82, 532.29) mm, rotated rx -180 ry 0 rz -88.32 deg; joints [5.415, -23.987, -48.803, 14.109, -20.983, -18.234]
  MoveL 440 to (110.97, 1705.5, 532.29) mm, rotated rx -180 ry 0 rz -88.32 deg; joints [5.362, -23.826, -48.69, 14.04, -20.926, -18.136]
  MoveL 441 to (110.01, 1708.18, 532.29) mm, rotated rx -180 ry 0 rz -88.32 deg; joints [5.31, -23.665, -48.576, 13.971, -20.868, -18.039]
  MoveL 442 to (109.05, 1710.86, 532.29) mm, rotated rx -180 ry 0 rz -88.32 deg; joints [5.258, -23.504, -48.462, 13.902, -20.812, -17.942]
  MoveL 443 to (108.1, 1713.55, 532.29) mm, rotated rx -180 ry 0 rz -88.32 deg; joints [5.207, -23.344, -48.348, 13.834, -20.755, -17.847]
  MoveL 444 to (107.15, 1716.24, 532.29) mm, rotated rx 180 ry 0 rz -88.32 deg; joints [5.156, -23.183, -48.234, 13.767, -20.7, -17.751]
  MoveL 445 to (106.22, 1718.93, 532.29) mm, rotated rx -180 ry 0 rz -88.32 deg; joints [5.106, -23.022, -48.119, 13.7, -20.644, -17.657]
  MoveL 446 to (105.29, 1721.62, 532.29) mm, rotated rx -180 ry 0 rz -88.32 deg; joints [5.056, -22.862, -48.004, 13.633, -20.589, -17.563]
  MoveL 447 to (104.37, 1724.32, 532.29) mm, rotated rx -180 ry 0 rz -88.32 deg; joints [5.007, -22.701, -47.889, 13.567, -20.535, -17.47]
  MoveL 448 to (103.45, 1727.02, 532.29) mm, rotated rx 180 ry 0 rz -88.32 deg; joints [4.958, -22.541, -47.774, 13.501, -20.481, -17.378]
  MoveL 449 to (102.55, 1729.72, 532.29) mm, rotated rx 180 ry 0 rz -88.32 deg; joints [4.91, -22.381, -47.658, 13.436, -20.427, -17.286]
  MoveL 450 to (101.65, 1732.43, 532.29) mm, rotated rx -180 ry 0 rz -88.32 deg; joints [4.862, -22.22, -47.542, 13.371, -20.374, -17.195]
  MoveL 451 to (100.76, 1735.13, 532.29) mm, rotated rx -180 ry 0 rz -88.32 deg; joints [4.815, -22.06, -47.426, 13.307, -20.321, -17.105]
  MoveL 452 to (99.87, 1737.84, 532.29) mm, rotated rx 180 ry 0 rz -88.32 deg; joints [4.768, -21.9, -47.309, 13.243, -20.269, -17.015]
  MoveL 453 to (99, 1740.55, 532.29) mm, rotated rx 180 ry 0 rz -88.32 deg; joints [4.722, -21.74, -47.193, 13.179, -20.217, -16.926]
  MoveL 454 to (98.13, 1743.27, 532.29) mm, rotated rx -180 ry 0 rz -88.32 deg; joints [4.676, -21.58, -47.076, 13.116, -20.165, -16.838]
  MoveL 455 to (97.27, 1745.98, 532.29) mm, rotated rx -180 ry 0 rz -88.32 deg; joints [4.63, -21.42, -46.959, 13.053, -20.114, -16.75]
  MoveL 456 to (96.42, 1748.7, 532.29) mm, rotated rx -180 ry 0 rz -88.32 deg; joints [4.586, -21.26, -46.841, 12.991, -20.064, -16.663]
  MoveL 457 to (95.57, 1751.43, 532.29) mm, rotated rx 180 ry 0 rz -88.32 deg; joints [4.541, -21.1, -46.723, 12.929, -20.014, -16.577]
  MoveL 458 to (94.73, 1754.15, 532.29) mm, rotated rx 180 ry 0 rz -88.32 deg; joints [4.497, -20.94, -46.606, 12.868, -19.964, -16.492]
  MoveL 459 to (93.9, 1756.88, 532.29) mm, rotated rx -180 ry 0 rz -88.32 deg; joints [4.454, -20.78, -46.487, 12.807, -19.915, -16.407]
  MoveL 460 to (93.08, 1759.6, 532.29) mm, rotated rx -180 ry 0 rz -88.32 deg; joints [4.411, -20.621, -46.369, 12.747, -19.866, -16.323]
  MoveL 461 to (92.27, 1762.34, 532.29) mm, rotated rx -180 ry 0 rz -88.32 deg; joints [4.369, -20.461, -46.25, 12.687, -19.818, -16.24]
  MoveL 462 to (91.46, 1765.07, 532.29) mm, rotated rx -180 ry 0 rz -88.32 deg; joints [4.327, -20.301, -46.132, 12.628, -19.77, -16.157]
  MoveL 463 to (90.66, 1767.8, 532.29) mm, rotated rx -180 ry 0 rz -88.32 deg; joints [4.285, -20.142, -46.012, 12.569, -19.722, -16.075]
  MoveL 464 to (89.87, 1770.54, 532.29) mm, rotated rx -180 ry 0 rz -88.32 deg; joints [4.244, -19.983, -45.893, 12.51, -19.675, -15.994]
  MoveL 465 to (89.08, 1773.28, 532.29) mm, rotated rx -180 ry 0 rz -88.32 deg; joints [4.204, -19.823, -45.774, 12.452, -19.629, -15.914]
  MoveL 466 to (88.31, 1776.02, 532.29) mm, rotated rx 180 ry 0 rz -88.32 deg; joints [4.163, -19.664, -45.654, 12.395, -19.582, -15.834]
  MoveL 467 to (87.54, 1778.77, 532.29) mm, rotated rx 180 ry 0 rz -88.32 deg; joints [4.124, -19.505, -45.534, 12.338, -19.537, -15.755]
  MoveL 468 to (86.78, 1781.51, 532.29) mm, rotated rx 180 ry 0 rz -88.32 deg; joints [4.085, -19.346, -45.414, 12.281, -19.491, -15.677]
  MoveL 469 to (86.02, 1784.26, 532.29) mm, rotated rx 180 ry 0 rz -88.32 deg; joints [4.046, -19.187, -45.293, 12.225, -19.446, -15.6]
  MoveL 470 to (85.28, 1787.01, 532.29) mm, rotated rx -180 ry 0 rz -88.32 deg; joints [4.008, -19.029, -45.172, 12.17, -19.402, -15.523]
  MoveL 471 to (84.54, 1789.77, 532.29) mm, rotated rx 180 ry 0 rz -88.32 deg; joints [3.97, -18.87, -45.052, 12.114, -19.358, -15.447]
  MoveL 472 to (83.81, 1792.52, 532.29) mm, rotated rx -180 ry 0 rz -88.32 deg; joints [3.933, -18.711, -44.93, 12.06, -19.314, -15.372]
  MoveL 473 to (83.09, 1795.28, 532.29) mm, rotated rx 180 ry 0 rz -88.32 deg; joints [3.896, -18.553, -44.809, 12.006, -19.271, -15.297]
  MoveL 474 to (82.37, 1798.04, 532.29) mm, rotated rx -180 ry 0 rz -88.32 deg; joints [3.859, -18.395, -44.688, 11.952, -19.228, -15.223]
  MoveL 475 to (81.67, 1800.8, 532.29) mm, rotated rx -180 ry 0 rz -88.32 deg; joints [3.823, -18.236, -44.566, 11.899, -19.186, -15.15]
  MoveL 476 to (80.97, 1803.56, 532.29) mm, rotated rx 180 ry 0 rz -88.32 deg; joints [3.788, -18.078, -44.444, 11.847, -19.144, -15.078]
  MoveL 477 to (80.28, 1806.33, 532.29) mm, rotated rx 180 ry 0 rz -88.32 deg; joints [3.752, -17.92, -44.322, 11.795, -19.102, -15.006]
  MoveL 478 to (79.59, 1809.09, 532.29) mm, rotated rx 180 ry 0 rz -88.32 deg; joints [3.718, -17.762, -44.199, 11.743, -19.061, -14.935]
  MoveL 479 to (78.92, 1811.86, 532.29) mm, rotated rx -180 ry 0 rz -88.32 deg; joints [3.684, -17.604, -44.077, 11.692, -19.02, -14.865]
  MoveL 480 to (78.25, 1814.63, 532.29) mm, rotated rx 180 ry 0 rz -88.32 deg; joints [3.65, -17.447, -43.954, 11.642, -18.98, -14.796]
  MoveL 481 to (77.59, 1817.4, 532.29) mm, rotated rx 180 ry 0 rz -88.32 deg; joints [3.616, -17.289, -43.831, 11.592, -18.94, -14.727]
  MoveL 482 to (76.94, 1820.18, 532.29) mm, rotated rx 180 ry 0 rz -88.32 deg; joints [3.583, -17.132, -43.707, 11.542, -18.901, -14.659]
  MoveL 483 to (76.29, 1822.95, 532.29) mm, rotated rx -180 ry 0 rz -88.32 deg; joints [3.551, -16.974, -43.584, 11.493, -18.862, -14.592]
  MoveL 484 to (75.65, 1825.73, 532.29) mm, rotated rx 180 ry 0 rz -88.32 deg; joints [3.519, -16.817, -43.46, 11.445, -18.823, -14.526]
  MoveL 485 to (75.03, 1828.51, 532.29) mm, rotated rx -180 ry 0 rz -88.32 deg; joints [3.487, -16.66, -43.337, 11.397, -18.785, -14.46]
  MoveL 486 to (74.4, 1831.29, 532.29) mm, rotated rx 180 ry 0 rz -88.32 deg; joints [3.456, -16.503, -43.212, 11.35, -18.747, -14.395]
  MoveL 487 to (73.79, 1834.07, 532.29) mm, rotated rx -180 ry 0 rz -88.32 deg; joints [3.425, -16.346, -43.088, 11.303, -18.71, -14.331]
  MoveL 488 to (73.18, 1836.86, 532.29) mm, rotated rx -180 ry 0 rz -88.32 deg; joints [3.395, -16.189, -42.964, 11.256, -18.673, -14.268]
  MoveL 489 to (72.59, 1839.65, 532.29) mm, rotated rx -180 ry 0 rz -88.32 deg; joints [3.365, -16.033, -42.839, 11.211, -18.636, -14.205]
  MoveL 490 to (72, 1842.43, 532.29) mm, rotated rx 180 ry 0 rz -88.32 deg; joints [3.335, -15.876, -42.714, 11.165, -18.6, -14.144]
  MoveL 491 to (71.41, 1845.22, 532.29) mm, rotated rx 180 ry 0 rz -88.32 deg; joints [3.306, -15.72, -42.589, 11.121, -18.564, -14.082]
  MoveL 492 to (70.84, 1848.02, 532.29) mm, rotated rx -180 ry 0 rz -88.32 deg; joints [3.277, -15.563, -42.464, 11.076, -18.529, -14.022]
  MoveL 493 to (70.27, 1850.81, 532.29) mm, rotated rx -180 ry 0 rz -88.32 deg; joints [3.249, -15.407, -42.338, 11.033, -18.494, -13.963]
  MoveL 494 to (69.71, 1853.6, 532.29) mm, rotated rx 180 ry 0 rz -88.32 deg; joints [3.221, -15.251, -42.213, 10.99, -18.459, -13.904]
  MoveL 495 to (69.16, 1856.4, 532.29) mm, rotated rx -180 ry 0 rz -88.32 deg; joints [3.193, -15.095, -42.087, 10.947, -18.425, -13.846]
  MoveL 496 to (68.62, 1859.2, 532.29) mm, rotated rx 180 ry 0 rz -88.32 deg; joints [3.166, -14.94, -41.961, 10.905, -18.391, -13.789]
  MoveL 497 to (68.09, 1862, 532.29) mm, rotated rx -180 ry 0 rz -88.32 deg; joints [3.14, -14.784, -41.835, 10.864, -18.358, -13.732]
  MoveL 498 to (67.56, 1864.8, 532.29) mm, rotated rx -180 ry 0 rz -88.32 deg; joints [3.113, -14.629, -41.708, 10.823, -18.325, -13.676]
  MoveL 499 to (67.04, 1867.6, 532.29) mm, rotated rx -180 ry 0 rz -88.32 deg; joints [3.087, -14.473, -41.582, 10.782, -18.292, -13.621]
  MoveL 500 to (66.53, 1870.4, 532.29) mm, rotated rx 180 ry 0 rz -88.32 deg; joints [3.062, -14.318, -41.455, 10.743, -18.26, -13.567]
  MoveL 501 to (66.02, 1873.21, 532.29) mm, rotated rx 180 ry 0 rz -88.32 deg; joints [3.037, -14.163, -41.328, 10.703, -18.228, -13.514]
  MoveL 502 to (65.53, 1876.01, 532.29) mm, rotated rx 180 ry 0 rz -88.32 deg; joints [3.012, -14.008, -41.201, 10.664, -18.197, -13.461]
  MoveL 503 to (65.04, 1878.82, 532.29) mm, rotated rx 180 ry 0 rz -88.32 deg; joints [2.988, -13.853, -41.074, 10.626, -18.166, -13.409]
  MoveL 504 to (64.56, 1881.63, 532.29) mm, rotated rx -180 ry 0 rz -88.32 deg; joints [2.964, -13.698, -40.946, 10.589, -18.135, -13.358]
  MoveL 505 to (64.09, 1884.44, 532.29) mm, rotated rx -180 ry 0 rz -88.32 deg; joints [2.94, -13.544, -40.818, 10.552, -18.105, -13.308]
  MoveL 506 to (63.62, 1887.25, 532.29) mm, rotated rx -180 ry 0 rz -88.32 deg; joints [2.917, -13.389, -40.691, 10.515, -18.075, -13.258]
  MoveL 507 to (63.17, 1890.07, 532.29) mm, rotated rx -180 ry 0 rz -88.32 deg; joints [2.894, -13.235, -40.562, 10.479, -18.046, -13.209]
  MoveL 508 to (62.72, 1892.88, 532.29) mm, rotated rx -180 ry 0 rz -88.32 deg; joints [2.872, -13.081, -40.434, 10.444, -18.017, -13.161]
  MoveL 509 to (62.28, 1895.7, 532.29) mm, rotated rx 180 ry 0 rz -88.32 deg; joints [2.85, -12.927, -40.306, 10.409, -17.988, -13.114]
  MoveL 510 to (61.84, 1898.51, 532.29) mm, rotated rx -180 ry 0 rz -88.32 deg; joints [2.828, -12.773, -40.177, 10.375, -17.96, -13.067]
  MoveL 511 to (61.42, 1901.33, 532.29) mm, rotated rx -180 ry 0 rz -88.32 deg; joints [2.807, -12.62, -40.049, 10.341, -17.932, -13.022]
  MoveL 512 to (61, 1904.15, 532.29) mm, rotated rx 180 ry 0 rz -88.32 deg; joints [2.786, -12.466, -39.92, 10.308, -17.904, -12.977]
  MoveL 513 to (60.59, 1906.97, 532.29) mm, rotated rx -180 ry 0 rz -88.32 deg; joints [2.765, -12.313, -39.791, 10.275, -17.877, -12.932]
  MoveL 514 to (60.19, 1909.79, 532.29) mm, rotated rx -180 ry 0 rz -88.32 deg; joints [2.745, -12.159, -39.661, 10.243, -17.85, -12.889]
  MoveL 515 to (59.8, 1912.61, 532.29) mm, rotated rx -180 ry 0 rz -88.32 deg; joints [2.725, -12.006, -39.532, 10.212, -17.824, -12.846]
  MoveL 516 to (59.41, 1915.44, 532.29) mm, rotated rx -180 ry 0 rz -88.32 deg; joints [2.706, -11.853, -39.402, 10.181, -17.798, -12.804]
  MoveL 517 to (59.03, 1918.26, 532.29) mm, rotated rx -180 ry 0 rz -88.32 deg; joints [2.687, -11.7, -39.272, 10.15, -17.772, -12.763]
  MoveL 518 to (58.67, 1921.09, 532.29) mm, rotated rx -180 ry 0 rz -88.32 deg; joints [2.668, -11.548, -39.143, 10.12, -17.747, -12.723]
  MoveL 519 to (58.3, 1923.91, 532.29) mm, rotated rx 180 ry 0 rz -88.32 deg; joints [2.65, -11.395, -39.012, 10.091, -17.722, -12.683]
  MoveL 520 to (57.95, 1926.74, 532.29) mm, rotated rx -180 ry 0 rz -88.32 deg; joints [2.632, -11.243, -38.882, 10.063, -17.697, -12.644]
  MoveL 521 to (57.6, 1929.57, 532.29) mm, rotated rx 180 ry 0 rz -88.32 deg; joints [2.614, -11.091, -38.752, 10.034, -17.673, -12.606]
  MoveL 522 to (57.27, 1932.4, 532.29) mm, rotated rx -180 ry 0 rz -88.32 deg; joints [2.597, -10.938, -38.621, 10.007, -17.649, -12.569]
  MoveL 523 to (56.94, 1935.23, 532.29) mm, rotated rx 180 ry 0 rz -88.32 deg; joints [2.58, -10.786, -38.49, 9.98, -17.626, -12.532]
  MoveL 524 to (56.61, 1938.06, 532.29) mm, rotated rx 180 ry 0 rz -88.32 deg; joints [2.564, -10.635, -38.359, 9.954, -17.603, -12.497]
  MoveL 525 to (56.3, 1940.9, 532.29) mm, rotated rx -180 ry 0 rz -88.32 deg; joints [2.547, -10.483, -38.228, 9.928, -17.58, -12.462]
  MoveL 526 to (55.99, 1943.73, 532.29) mm, rotated rx -180 ry 0 rz -88.32 deg; joints [2.531, -10.332, -38.097, 9.902, -17.558, -12.427]
  MoveL 527 to (55.7, 1946.56, 532.29) mm, rotated rx 180 ry 0 rz -88.32 deg; joints [2.516, -10.18, -37.966, 9.878, -17.536, -12.394]
  MoveL 528 to (55.41, 1949.4, 532.29) mm, rotated rx 180 ry 0 rz -88.32 deg; joints [2.501, -10.029, -37.834, 9.854, -17.514, -12.361]
  MoveL 529 to (55.12, 1952.23, 532.29) mm, rotated rx -180 ry 0 rz -88.32 deg; joints [2.486, -9.878, -37.702, 9.83, -17.493, -12.329]
  MoveL 530 to (54.85, 1955.07, 532.29) mm, rotated rx -180 ry 0 rz -88.32 deg; joints [2.471, -9.727, -37.571, 9.807, -17.472, -12.298]
  MoveL 531 to (54.58, 1957.91, 532.29) mm, rotated rx 180 ry 0 rz -88.32 deg; joints [2.457, -9.576, -37.439, 9.785, -17.451, -12.268]
  MoveL 532 to (54.33, 1960.75, 532.29) mm, rotated rx -180 ry 0 rz -88.32 deg; joints [2.444, -9.426, -37.306, 9.763, -17.431, -12.238]
  MoveL 533 to (54.07, 1963.59, 532.29) mm, rotated rx -180 ry 0 rz -88.32 deg; joints [2.43, -9.275, -37.174, 9.741, -17.411, -12.209]
  MoveL 534 to (53.83, 1966.43, 532.29) mm, rotated rx 180 ry 0 rz -88.32 deg; joints [2.417, -9.125, -37.042, 9.721, -17.392, -12.181]
  MoveL 535 to (53.6, 1969.27, 532.29) mm, rotated rx 180 ry 0 rz -88.32 deg; joints [2.404, -8.975, -36.909, 9.7, -17.372, -12.153]
  MoveL 536 to (53.37, 1972.11, 532.29) mm, rotated rx 180 ry 0 rz -88.32 deg; joints [2.392, -8.825, -36.776, 9.681, -17.354, -12.127]
  MoveL 537 to (53.15, 1974.95, 532.29) mm, rotated rx -180 ry 0 rz -88.32 deg; joints [2.38, -8.675, -36.643, 9.662, -17.335, -12.101]
  MoveL 538 to (52.94, 1977.79, 532.29) mm, rotated rx -180 ry 0 rz -88.32 deg; joints [2.368, -8.525, -36.51, 9.643, -17.317, -12.075]
  MoveL 539 to (52.74, 1980.63, 532.29) mm, rotated rx -180 ry 0 rz -88.32 deg; joints [2.356, -8.376, -36.377, 9.625, -17.299, -12.051]
  MoveL 540 to (52.55, 1983.48, 532.29) mm, rotated rx 180 ry 0 rz -88.32 deg; joints [2.345, -8.226, -36.243, 9.608, -17.282, -12.027]
  MoveL 541 to (52.36, 1986.32, 532.29) mm, rotated rx -180 ry 0 rz -88.32 deg; joints [2.334, -8.077, -36.11, 9.591, -17.265, -12.004]
  MoveL 542 to (52.18, 1989.16, 532.29) mm, rotated rx -180 ry 0 rz -88.32 deg; joints [2.324, -7.928, -35.976, 9.575, -17.248, -11.982]
  MoveL 543 to (52.01, 1992.01, 532.29) mm, rotated rx -180 ry 0 rz -88.32 deg; joints [2.314, -7.779, -35.842, 9.559, -17.232, -11.961]
  MoveL 544 to (51.85, 1994.85, 532.29) mm, rotated rx -180 ry 0 rz -88.32 deg; joints [2.304, -7.631, -35.708, 9.544, -17.216, -11.94]
  MoveL 545 to (51.69, 1997.7, 532.29) mm, rotated rx 180 ry 0 rz -88.32 deg; joints [2.294, -7.482, -35.574, 9.529, -17.2, -11.92]
  MoveL 546 to (51.55, 2000.55, 532.29) mm, rotated rx -180 ry 0 rz -88.32 deg; joints [2.285, -7.334, -35.44, 9.515, -17.185, -11.901]
  MoveL 547 to (51.41, 2003.39, 532.29) mm, rotated rx -180 ry 0 rz -88.32 deg; joints [2.276, -7.185, -35.306, 9.502, -17.17, -11.882]
  MoveL 548 to (51.28, 2006.24, 532.29) mm, rotated rx 180 ry 0 rz -88.32 deg; joints [2.267, -7.037, -35.171, 9.489, -17.155, -11.864]
  MoveL 549 to (51.15, 2009.09, 532.29) mm, rotated rx 180 ry 0 rz -88.32 deg; joints [2.259, -6.889, -35.037, 9.477, -17.141, -11.847]
  MoveL 550 to (51.04, 2011.93, 532.29) mm, rotated rx 180 ry 0 rz -88.32 deg; joints [2.251, -6.741, -34.902, 9.465, -17.127, -11.831]
  MoveL 551 to (50.93, 2014.78, 532.29) mm, rotated rx 180 ry 0 rz -88.32 deg; joints [2.243, -6.594, -34.767, 9.454, -17.113, -11.816]
  MoveL 552 to (50.83, 2017.63, 532.29) mm, rotated rx -180 ry 0 rz -88.32 deg; joints [2.236, -6.446, -34.632, 9.443, -17.1, -11.801]
  MoveL 553 to (50.74, 2020.48, 532.29) mm, rotated rx 180 ry 0 rz -88.32 deg; joints [2.229, -6.299, -34.497, 9.433, -17.087, -11.787]
  MoveL 554 to (50.66, 2023.33, 532.29) mm, rotated rx -180 ry 0 rz -88.32 deg; joints [2.222, -6.152, -34.361, 9.423, -17.074, -11.773]
  MoveL 555 to (50.58, 2026.18, 532.29) mm, rotated rx 180 ry 0 rz -88.32 deg; joints [2.216, -6.005, -34.226, 9.414, -17.062, -11.76]
  MoveL 556 to (50.52, 2029.02, 532.29) mm, rotated rx 180 ry 0 rz -88.32 deg; joints [2.21, -5.858, -34.09, 9.405, -17.05, -11.748]
  MoveL 557 to (50.46, 2031.87, 532.29) mm, rotated rx 180 ry 0 rz -88.32 deg; joints [2.204, -5.711, -33.954, 9.397, -17.038, -11.737]
  MoveL 558 to (50.41, 2034.72, 532.29) mm, rotated rx -180 ry 0 rz -88.32 deg; joints [2.198, -5.564, -33.818, 9.39, -17.027, -11.727]
  MoveL 559 to (50.37, 2037.57, 532.29) mm, rotated rx -180 ry 0 rz -88.32 deg; joints [2.193, -5.418, -33.682, 9.383, -17.016, -11.717]
  MoveL 560 to (50.33, 2040.42, 532.29) mm, rotated rx -180 ry 0 rz -88.32 deg; joints [2.188, -5.272, -33.546, 9.377, -17.005, -11.708]
  MoveL 561 to (50.3, 2043.27, 532.29) mm, rotated rx -180 ry 0 rz -88.32 deg; joints [2.183, -5.126, -33.41, 9.371, -16.995, -11.699]
  MoveL 562 to (50.28, 2046.12, 532.29) mm, rotated rx -180 ry 0 rz -88.32 deg; joints [2.179, -4.98, -33.274, 9.365, -16.985, -11.691]
  MoveL 563 to (50.27, 2048.97, 532.29) mm, rotated rx 180 ry 0 rz -88.32 deg; joints [2.175, -4.834, -33.137, 9.361, -16.975, -11.684]
  MoveL 564 to (50.27, 2051.82, 532.29) mm, rotated rx -180 ry 0 rz -88.32 deg; joints [2.171, -4.688, -33, 9.356, -16.965, -11.678]
  MoveL 565 to (50.28, 2054.67, 532.29) mm, rotated rx 180 ry 0 rz -88.32 deg; joints [2.167, -4.543, -32.864, 9.353, -16.956, -11.672]
  MoveL 566 to (50.29, 2057.52, 532.29) mm, rotated rx 180 ry 0 rz -88.32 deg; joints [2.164, -4.397, -32.727, 9.349, -16.948, -11.667]
  MoveL 567 to (50.31, 2060.37, 532.29) mm, rotated rx -180 ry 0 rz -88.32 deg; joints [2.161, -4.252, -32.59, 9.347, -16.939, -11.663]
  MoveL 568 to (50.34, 2063.22, 532.29) mm, rotated rx 180 ry 0 rz -88.32 deg; joints [2.158, -4.107, -32.452, 9.344, -16.931, -11.659]
  MoveL 569 to (50.38, 2066.07, 532.29) mm, rotated rx 180 ry 0 rz -88.32 deg; joints [2.156, -3.962, -32.315, 9.343, -16.923, -11.657]
  MoveL 570 to (50.42, 2068.92, 532.29) mm, rotated rx -180 ry 0 rz -88.32 deg; joints [2.154, -3.817, -32.178, 9.342, -16.916, -11.654]
  MoveL 571 to (50.47, 2071.77, 532.29) mm, rotated rx -180 ry 0 rz -88.32 deg; joints [2.152, -3.673, -32.04, 9.341, -16.908, -11.653]
  MoveL 572 to (50.54, 2074.62, 532.29) mm, rotated rx 180 ry 0 rz -88.32 deg; joints [2.151, -3.529, -31.902, 9.341, -16.902, -11.652]
  MoveL 573 to (50.6, 2077.47, 532.29) mm, rotated rx -180 ry 0 rz -88.32 deg; joints [2.149, -3.384, -31.765, 9.341, -16.895, -11.652]
  MoveL 574 to (50.68, 2080.32, 532.29) mm, rotated rx -180 ry 0 rz -88.32 deg; joints [2.148, -3.24, -31.627, 9.342, -16.889, -11.652]
  MoveL 575 to (50.77, 2083.16, 532.29) mm, rotated rx 180 ry 0 rz -88.32 deg; joints [2.148, -3.096, -31.489, 9.344, -16.883, -11.653]
  MoveL 576 to (50.86, 2086.01, 532.29) mm, rotated rx -180 ry 0 rz -88.32 deg; joints [2.147, -2.952, -31.351, 9.346, -16.877, -11.655]
  MoveL 577 to (50.96, 2088.86, 532.29) mm, rotated rx 180 ry 0 rz -88.32 deg; joints [2.147, -2.809, -31.212, 9.348, -16.872, -11.657]
  MoveL 578 to (51.07, 2091.71, 532.29) mm, rotated rx -180 ry 0 rz -88.32 deg; joints [2.147, -2.665, -31.074, 9.351, -16.867, -11.66]
  MoveL 579 to (51.19, 2094.56, 532.29) mm, rotated rx -180 ry 0 rz -88.32 deg; joints [2.147, -2.522, -30.935, 9.354, -16.862, -11.664]
  MoveL 580 to (51.31, 2097.4, 532.29) mm, rotated rx -180 ry 0 rz -88.32 deg; joints [2.148, -2.379, -30.797, 9.358, -16.858, -11.669]
  MoveL 581 to (51.44, 2100.25, 532.29) mm, rotated rx -180 ry 0 rz -88.32 deg; joints [2.149, -2.236, -30.658, 9.363, -16.854, -11.674]
  MoveL 582 to (51.59, 2103.1, 532.29) mm, rotated rx -180 ry 0 rz -88.32 deg; joints [2.15, -2.093, -30.519, 9.367, -16.85, -11.679]
  MoveL 583 to (51.73, 2105.94, 532.29) mm, rotated rx -180 ry 0 rz -88.32 deg; joints [2.151, -1.95, -30.38, 9.373, -16.846, -11.685]
  MoveL 584 to (51.89, 2108.79, 532.29) mm, rotated rx -180 ry 0 rz -88.32 deg; joints [2.153, -1.808, -30.241, 9.379, -16.843, -11.692]
  MoveL 585 to (52.06, 2111.63, 532.29) mm, rotated rx -180 ry 0 rz -88.32 deg; joints [2.155, -1.665, -30.102, 9.385, -16.84, -11.7]
  MoveL 586 to (52.23, 2114.48, 532.29) mm, rotated rx 180 ry 0 rz -88.32 deg; joints [2.157, -1.523, -29.963, 9.392, -16.838, -11.708]
  MoveL 587 to (52.41, 2117.32, 532.29) mm, rotated rx 180 ry 0 rz -88.32 deg; joints [2.159, -1.381, -29.823, 9.399, -16.835, -11.717]
  MoveL 588 to (52.6, 2120.17, 532.29) mm, rotated rx 180 ry 0 rz -88.32 deg; joints [2.162, -1.239, -29.684, 9.407, -16.833, -11.726]
  MoveL 589 to (52.8, 2123.01, 532.29) mm, rotated rx -180 ry 0 rz -88.32 deg; joints [2.165, -1.097, -29.544, 9.415, -16.832, -11.736]
  MoveL 590 to (53, 2125.85, 532.29) mm, rotated rx 180 ry 0 rz -88.32 deg; joints [2.168, -0.955, -29.404, 9.424, -16.83, -11.747]
  MoveL 591 to (53.21, 2128.69, 532.29) mm, rotated rx 180 ry 0 rz -88.32 deg; joints [2.172, -0.814, -29.264, 9.433, -16.829, -11.758]
  MoveL 592 to (53.43, 2131.53, 532.29) mm, rotated rx 180 ry 0 rz -88.32 deg; joints [2.175, -0.673, -29.124, 9.442, -16.828, -11.77]
  MoveL 593 to (53.66, 2134.37, 532.29) mm, rotated rx 180 ry 0 rz -88.32 deg; joints [2.179, -0.531, -28.984, 9.452, -16.828, -11.783]
  MoveL 594 to (53.9, 2137.22, 532.29) mm, rotated rx 180 ry 0 rz -88.32 deg; joints [2.184, -0.39, -28.844, 9.463, -16.828, -11.796]
  MoveL 595 to (54.14, 2140.05, 532.29) mm, rotated rx -180 ry 0 rz -88.32 deg; joints [2.188, -0.249, -28.704, 9.474, -16.828, -11.809]
  MoveL 596 to (54.4, 2142.89, 532.29) mm, rotated rx 180 ry 0 rz -88.32 deg; joints [2.193, -0.109, -28.563, 9.485, -16.828, -11.824]
  MoveL 597 to (54.66, 2145.73, 532.29) mm, rotated rx 180 ry 0 rz -88.32 deg; joints [2.198, 0.032, -28.423, 9.497, -16.829, -11.838]
  MoveL 598 to (54.93, 2148.57, 532.29) mm, rotated rx 180 ry 0 rz -88.32 deg; joints [2.203, 0.172, -28.282, 9.509, -16.83, -11.854]
  MoveL 599 to (55.2, 2151.4, 532.29) mm, rotated rx 180 ry 0 rz -88.32 deg; joints [2.208, 0.313, -28.141, 9.522, -16.831, -11.87]
  MoveL 600 to (55.49, 2154.24, 532.29) mm, rotated rx -180 ry 0 rz -88.32 deg; joints [2.214, 0.453, -28, 9.535, -16.832, -11.886]
  MoveL 601 to (55.78, 2157.07, 532.29) mm, rotated rx 180 ry 0 rz -88.32 deg; joints [2.22, 0.593, -27.86, 9.549, -16.834, -11.904]
  MoveL 602 to (56.08, 2159.91, 532.29) mm, rotated rx -180 ry 0 rz -88.32 deg; joints [2.226, 0.733, -27.718, 9.563, -16.836, -11.921]
  MoveL 603 to (56.39, 2162.74, 532.29) mm, rotated rx -180 ry 0 rz -88.32 deg; joints [2.232, 0.872, -27.577, 9.577, -16.839, -11.94]
  MoveL 604 to (56.7, 2165.57, 532.29) mm, rotated rx 180 ry 0 rz -88.32 deg; joints [2.239, 1.012, -27.436, 9.592, -16.841, -11.958]
  MoveL 605 to (57.03, 2168.41, 532.29) mm, rotated rx 180 ry 0 rz -88.32 deg; joints [2.246, 1.151, -27.295, 9.607, -16.844, -11.978]
  MoveL 606 to (57.36, 2171.24, 532.29) mm, rotated rx 180 ry 0 rz -88.32 deg; joints [2.253, 1.291, -27.153, 9.623, -16.847, -11.998]
  MoveL 607 to (57.7, 2174.07, 532.29) mm, rotated rx 180 ry 0 rz -88.32 deg; joints [2.26, 1.43, -27.012, 9.639, -16.851, -12.018]
  MoveL 608 to (58.05, 2176.89, 532.29) mm, rotated rx 180 ry 0 rz -88.32 deg; joints [2.268, 1.569, -26.87, 9.656, -16.855, -12.039]
  MoveL 609 to (58.4, 2179.72, 532.29) mm, rotated rx 180 ry 0 rz -88.32 deg; joints [2.276, 1.708, -26.728, 9.673, -16.859, -12.061]
